LIN {X 0,Y 412.505,Z 413.678,A -85,B 0,C 180,E1 -10494.601,E2 -10494.601} C_VEL
LIN {X 0,Y 412.069,Z 420.208,A -85,B 0,C 180,E1 -10498.081,E2 -10498.081} C_VEL
LIN {X 0,Y 411.614,Z 426.756,A -85,B 0,C 180,E1 -10501.44,E2 -10501.44} C_VEL
LIN {X 0,Y 411.176,Z 433.807,A -85,B 0,C 180,E1 -10504.945,E2 -10504.945} C_VEL
LIN {X 0,Y 410.804,Z 440.902,A -85,B 0,C 180,E1 -10508.419,E2 -10508.419} C_VEL
LIN {X 0,Y 410.512,Z 447.336,A -85,B 0,C 180,E1 -10511.535,E2 -10511.535} C_VEL
LIN {X 0,Y 410.473,Z 449.297,A -85,B 0,C 180,E1 -10512.42,E2 -10512.42} C_VEL
LIN {X 0,Y 412.911,Z 462.619,A -85,B 0,C 180,E1 -10512.936,E2 -10512.936} C_VEL
LIN {X 0,Y 414.711,Z 476.29,A -85,B 0,C 180,E1 -10513.666,E2 -10513.666} C_VEL
LIN {X 0,Y 414.65,Z 482.208,A -85,B 0,C 180,E1 -10514.024,E2 -10514.024} C_VEL
LIN {X 0,Y 413.868,Z 493.865,A -85,B 0,C 180,E1 -10514.865,E2 -10514.865} C_VEL
LIN {X 0,Y 413.021,Z 505.142,A -85,B 0,C 180,E1 -10515.911,E2 -10515.911} C_VEL
LIN {X 0,Y 412.454,Z 514.201,A -85,B 0,C 180,E1 -10516.952,E2 -10516.952} C_VEL
LIN {X 0,Y 411.692,Z 523.047,A -85,B 0,C 180,E1 -10518.179,E2 -10518.179} C_VEL
LIN {X 0,Y 411.033,Z 531.675,A -85,B 0,C 180,E1 -10519.657,E2 -10519.657} C_VEL
LIN {X 0,Y 410.551,Z 538.575,A -85,B 0,C 180,E1 -10521.137,E2 -10521.137} C_VEL
LIN {X 0,Y 410.211,Z 544.105,A -85,B 0,C 180,E1 -10522.617,E2 -10522.617} C_VEL
LIN {X 0,Y 410.036,Z 548.444,A -85,B 0,C 180,E1 -10524.097,E2 -10524.097} C_VEL
LIN {X 0,Y 410.024,Z 550.743,A -85,B 0,C 180,E1 -10525.083,E2 -10525.083} C_VEL
LIN {X 0,Y 409.935,Z 552.604,A -85,B 0,C 180,E1 -10526.068,E2 -10526.068} C_VEL
LIN {X 0,Y 409.967,Z 554.999,A -85,B 0,C 180,E1 -10528.035,E2 -10528.035} C_VEL
LIN {X 0,Y 409.935,Z 555.607,A -85,B 0,C 180,E1 -10529.018,E2 -10529.018} C_VEL
LIN {X 0,Y 409.926,Z 555.822,A -85,B 0,C 180,E1 -10530,E2 -10530} C_VEL
LIN {X 0,Y 409.935,Z 555.605,A -85,B 0,C 180,E1 -10530.982,E2 -10530.982} C_VEL
LIN {X 0,Y 409.967,Z 554.998,A -85,B 0,C 180,E1 -10531.965,E2 -10531.965} C_VEL
LIN {X 0,Y 409.927,Z 553.999,A -85,B 0,C 180,E1 -10532.948,E2 -10532.948} C_VEL
LIN {X 0,Y 409.934,Z 552.601,A -85,B 0,C 180,E1 -10533.932,E2 -10533.932} C_VEL
LIN {X 0,Y 410.025,Z 549.663,A -85,B 0,C 180,E1 -10535.409,E2 -10535.409} C_VEL
LIN {X 0,Y 410.169,Z 545.685,A -85,B 0,C 180,E1 -10536.889,E2 -10536.889} C_VEL
LIN {X 0,Y 410.492,Z 539.57,A -85,B 0,C 180,E1 -10538.616,E2 -10538.616} C_VEL
LIN {X 0,Y 410.934,Z 532.89,A -85,B 0,C 180,E1 -10540.096,E2 -10540.096} C_VEL
LIN {X 0,Y 411.552,Z 524.604,A -85,B 0,C 180,E1 -10541.575,E2 -10541.575} C_VEL
LIN {X 0,Y 412.257,Z 516.113,A -85,B 0,C 180,E1 -10542.804,E2 -10542.804} C_VEL
LIN {X 0,Y 412.969,Z 506.149,A -85,B 0,C 180,E1 -10543.978,E2 -10543.978} C_VEL
LIN {X 0,Y 413.758,Z 495.239,A -85,B 0,C 180,E1 -10545.013,E2 -10545.013} C_VEL
LIN {X 0,Y 414.476,Z 483.946,A -85,B 0,C 180,E1 -10545.862,E2 -10545.862} C_VEL
LIN {X 0,Y 414.712,Z 476.208,A -85,B 0,C 180,E1 -10546.333,E2 -10546.333} C_VEL
LIN {X 0,Y 412.972,Z 463.345,A -85,B 0,C 180,E1 -10547.025,E2 -10547.025} C_VEL
LIN {X 0,Y 410.672,Z 450.687,A -85,B 0,C 180,E1 -10547.534,E2 -10547.534} C_VEL
LIN {X 0,Y 410.438,Z 449.15,A -85,B 0,C 180,E1 -10547.581,E2 -10547.581} C_VEL
LIN {X 0,Y 410.775,Z 441.97,A -85,B 0,C 180,E1 -10551.057,E2 -10551.057} C_VEL
LIN {X 0,Y 411.043,Z 435.469,A -85,B 0,C 180,E1 -10554.227,E2 -10554.227} C_VEL
LIN {X 0,Y 411.426,Z 428.914,A -85,B 0,C 180,E1 -10557.466,E2 -10557.466} C_VEL
LIN {X 0,Y 411.847,Z 423.443,A -85,B 0,C 180,E1 -10560.226,E2 -10560.226} C_VEL
LIN {X 0,Y 412.237,Z 417.454,A -85,B 0,C 180,E1 -10563.345,E2 -10563.345} C_VEL
LIN {X 0,Y 412.438,Z 412.57,A -85,B 0,C 180,E1 -10566.007,E2 -10566.007} C_VEL
LIN {X 0,Y 412.03,Z 408.565,A -85,B 0,C 180,E1 -10568.314,E2 -10568.314} C_VEL
LIN {X 0,Y 411.234,Z 404.262,A -85,B 0,C 180,E1 -10571.068,E2 -10571.068} C_VEL
LIN {X 0,Y 411.181,Z 404.267,A -85,B 0,C 180,E1 -10574.49,E2 -10574.49} C_VEL
LIN {X 0,Y 411.178,Z 404.264,A -85,B 0,C 180,E1 -10578.195,E2 -10578.195} C_VEL
LIN {X 0,Y 411.223,Z 404.263,A -85,B 0,C 180,E1 -10580.776,E2 -10580.776} C_VEL
LIN {X 0,Y 411.201,Z 404.264,A -85,B 0,C 180,E1 -10584.471,E2 -10584.471} C_VEL
LIN {X 0,Y 411.208,Z 404.265,A -85,B 0,C 180,E1 -10586.873,E2 -10586.873} C_VEL
LIN {X 0,Y 411.234,Z 404.261,A -85,B 0,C 180,E1 -10590.644,E2 -10590.644} C_VEL
LIN {X 0,Y 411.238,Z 404.257,A -85,B 0,C 180,E1 -10593.619,E2 -10593.619} C_VEL
LIN {X 0,Y 411.203,Z 404.265,A -85,B 0,C 180,E1 -10596.852,E2 -10596.852} C_VEL
LIN {X 0,Y 411.217,Z 404.262,A -85,B 0,C 180,E1 -10600.05,E2 -10600.05} C_VEL
LIN {X 0,Y 411.264,Z 404.255,A -85,B 0,C 180,E1 -10603.131,E2 -10603.131} C_VEL
LIN {X 0,Y 411.315,Z 404.25,A -85,B 0,C 180,E1 -10606.891,E2 -10606.891} C_VEL
LIN {X 0,Y 411.31,Z 404.253,A -85,B 0,C 180,E1 -10610.162,E2 -10610.162} C_VEL
LIN {X 0,Y 411.462,Z 404.23,A -85,B 0,C 180,E1 -10613.133,E2 -10613.133} C_VEL
LIN {X 0,Y 411.311,Z 404.248,A -85,B 0,C 180,E1 -10615.099,E2 -10615.099} C_VEL
LIN {X 0,Y 411.513,Z 404.226,A -85,B 0,C 180,E1 -10618.043,E2 -10618.043} C_VEL
LIN {X 0,Y 411.644,Z 404.21,A -85,B 0,C 180,E1 -10620,E2 -10620} C_VEL
LIN {X 0,Y 411.459,Z 404.23,A -85,B 0,C 180,E1 -10622.937,E2 -10622.937} C_VEL
LIN {X 0,Y 411.463,Z 404.23,A -85,B 0,C 180,E1 -10626.867,E2 -10626.867} C_VEL
LIN {X 0,Y 411.31,Z 404.251,A -85,B 0,C 180,E1 -10629.838,E2 -10629.838} C_VEL
LIN {X 0,Y 411.315,Z 404.247,A -85,B 0,C 180,E1 -10633.109,E2 -10633.109} C_VEL
LIN {X 0,Y 411.259,Z 404.255,A -85,B 0,C 180,E1 -10636.889,E2 -10636.889} C_VEL
LIN {X 0,Y 411.232,Z 404.262,A -85,B 0,C 180,E1 -10639.987,E2 -10639.987} C_VEL
LIN {X 0,Y 411.204,Z 404.262,A -85,B 0,C 180,E1 -10643.148,E2 -10643.148} C_VEL
LIN {X 0,Y 411.238,Z 404.257,A -85,B 0,C 180,E1 -10646.381,E2 -10646.381} C_VEL
LIN {X 0,Y 411.202,Z 404.266,A -85,B 0,C 180,E1 -10649.713,E2 -10649.713} C_VEL
LIN {X 0,Y 411.208,Z 404.264,A -85,B 0,C 180,E1 -10653.156,E2 -10653.156} C_VEL
LIN {X 0,Y 411.197,Z 404.262,A -85,B 0,C 180,E1 -10656.553,E2 -10656.553} C_VEL
LIN {X 0,Y 411.22,Z 404.262,A -85,B 0,C 180,E1 -10659.729,E2 -10659.729} C_VEL
LIN {X 0,Y 411.175,Z 404.269,A -85,B 0,C 180,E1 -10663.134,E2 -10663.134} C_VEL
LIN {X 0,Y 411.174,Z 404.267,A -85,B 0,C 180,E1 -10665.88,E2 -10665.88} C_VEL
LIN {X 0,Y 411.166,Z 404.268,A -85,B 0,C 180,E1 -10668.772,E2 -10668.772} C_VEL
LIN {X 0,Y 411.203,Z 404.266,A -85,B 0,C 180,E1 -10671.832,E2 -10671.832} C_VEL
LIN {X 0,Y 411.062,Z 404.442,A -85,B 0,C 180,E1 -10674.458,E2 -10674.458} C_VEL
LIN {X 0,Y 411.062,Z 407.378,A -85,B 0,C 180,E1 -10676.905,E2 -10676.905} C_VEL
LIN {X 0,Y 410.847,Z 411.553,A -85,B 0,C 180,E1 -10680.259,E2 -10680.259} C_VEL
LIN {X 0,Y 410.656,Z 415.795,A -85,B 0,C 180,E1 -10683.579,E2 -10683.579} C_VEL
LIN {X 0,Y 410.558,Z 418.639,A -85,B 0,C 180,E1 -10685.743,E2 -10685.743} C_VEL
LIN {X 0,Y 410.376,Z 422.946,A -85,B 0,C 180,E1 -10688.922,E2 -10688.922} C_VEL
LIN {X 0,Y 410.291,Z 427.335,A -85,B 0,C 180,E1 -10692.042,E2 -10692.042} C_VEL
LIN {X 0,Y 410.305,Z 428.198,A -85,B 0,C 180,E1 -10692.495,E2 -10692.495} C_VEL
LIN {X 0,Y 413.403,Z 441.217,A -85,B 0,C 180,E1 -10693.063,E2 -10693.063} C_VEL
LIN {X 0,Y 415.297,Z 451.396,A -85,B 0,C 180,E1 -10693.628,E2 -10693.628} C_VEL
LIN {X 0,Y 414.751,Z 463.825,A -85,B 0,C 180,E1 -10694.395,E2 -10694.395} C_VEL
LIN {X 0,Y 414.051,Z 474.588,A -85,B 0,C 180,E1 -10695.25,E2 -10695.25} C_VEL
LIN {X 0,Y 413.366,Z 485.554,A -85,B 0,C 180,E1 -10696.355,E2 -10696.355} C_VEL
LIN {X 0,Y 412.581,Z 494.46,A -85,B 0,C 180,E1 -10697.456,E2 -10697.456} C_VEL
LIN {X 0,Y 412.005,Z 502.624,A -85,B 0,C 180,E1 -10698.687,E2 -10698.687} C_VEL
LIN {X 0,Y 411.336,Z 510.624,A -85,B 0,C 180,E1 -10700.162,E2 -10700.162} C_VEL
LIN {X 0,Y 410.76,Z 517.048,A -85,B 0,C 180,E1 -10701.638,E2 -10701.638} C_VEL
LIN {X 0,Y 410.435,Z 522.648,A -85,B 0,C 180,E1 -10703.293,E2 -10703.293} C_VEL
LIN {X 0,Y 410.165,Z 527.155,A -85,B 0,C 180,E1 -10705.085,E2 -10705.085} C_VEL
LIN {X 0,Y 410.058,Z 529.016,A -85,B 0,C 180,E1 -10706.069,E2 -10706.069} C_VEL
LIN {X 0,Y 410.06,Z 530.414,A -85,B 0,C 180,E1 -10707.053,E2 -10707.053} C_VEL
LIN {X 0,Y 410.013,Z 531.41,A -85,B 0,C 180,E1 -10708.036,E2 -10708.036} C_VEL
LIN {X 0,Y 409.927,Z 532.258,A -85,B 0,C 180,E1 -10710,E2 -10710} C_VEL
LIN {X 0,Y 409.939,Z 532.07,A -85,B 0,C 180,E1 -10710.982,E2 -10710.982} C_VEL
LIN {X 0,Y 410.013,Z 531.484,A -85,B 0,C 180,E1 -10711.965,E2 -10711.965} C_VEL
LIN {X 0,Y 410.056,Z 530.518,A -85,B 0,C 180,E1 -10712.947,E2 -10712.947} C_VEL
LIN {X 0,Y 410.046,Z 529.165,A -85,B 0,C 180,E1 -10713.931,E2 -10713.931} C_VEL
LIN {X 0,Y 410.272,Z 526.298,A -85,B 0,C 180,E1 -10715.406,E2 -10715.406} C_VEL
LIN {X 0,Y 410.436,Z 522.415,A -85,B 0,C 180,E1 -10716.884,E2 -10716.884} C_VEL
LIN {X 0,Y 410.757,Z 517.403,A -85,B 0,C 180,E1 -10718.363,E2 -10718.363} C_VEL
LIN {X 0,Y 410.982,Z 514.645,A -85,B 0,C 180,E1 -10719.047,E2 -10719.047} C_VEL
LIN {X 0,Y 410.578,Z 511.665,A -85,B 0,C 180,E1 -10719.758,E2 -10719.758} C_VEL
LIN {X 0,Y 408.165,Z 506.457,A -85,B 0,C 180,E1 -10720.893,E2 -10720.893} C_VEL
LIN {X 0,Y 405.817,Z 500.596,A -85,B 0,C 180,E1 -10721.972,E2 -10721.972} C_VEL
LIN {X 0,Y 405.513,Z 496.593,A -85,B 0,C 180,E1 -10722.586,E2 -10722.586} C_VEL
LIN {X 0,Y 406.42,Z 486.565,A -85,B 0,C 180,E1 -10723.883,E2 -10723.883} C_VEL
LIN {X 0,Y 407.086,Z 475.827,A -85,B 0,C 180,E1 -10725.009,E2 -10725.009} C_VEL
LIN {X 0,Y 407.854,Z 465.354,A -85,B 0,C 180,E1 -10725.876,E2 -10725.876} C_VEL
LIN {X 0,Y 408.536,Z 453.254,A -85,B 0,C 180,E1 -10726.654,E2 -10726.654} C_VEL
LIN {X 0,Y 406.632,Z 442.722,A -85,B 0,C 180,E1 -10727.27,E2 -10727.27} C_VEL
LIN {X 0,Y 403.464,Z 429.728,A -85,B 0,C 180,E1 -10727.873,E2 -10727.873} C_VEL
LIN {X 0,Y 403.203,Z 428.147,A -85,B 0,C 180,E1 -10727.947,E2 -10727.947} C_VEL
LIN {X 0,Y 403.303,Z 424.709,A -85,B 0,C 180,E1 -10730.397,E2 -10730.397} C_VEL
LIN {X 0,Y 403.447,Z 420.388,A -85,B 0,C 180,E1 -10733.619,E2 -10733.619} C_VEL
LIN {X 0,Y 403.665,Z 416.097,A -85,B 0,C 180,E1 -10736.915,E2 -10736.915} C_VEL
LIN {X 0,Y 403.841,Z 411.84,A -85,B 0,C 180,E1 -10740.311,E2 -10740.311} C_VEL
LIN {X 0,Y 404.038,Z 407.549,A -85,B 0,C 180,E1 -10743.823,E2 -10743.823} C_VEL
LIN {X 0,Y 404.047,Z 405.966,A -85,B 0,C 180,E1 -10745.162,E2 -10745.162} C_VEL
LIN {X 0,Y 404.083,Z 405.153,A -85,B 0,C 180,E1 -10746.253,E2 -10746.253} C_VEL
LIN {X 0,Y 404.155,Z 405.145,A -85,B 0,C 180,E1 -10748.757,E2 -10748.757} C_VEL
LIN {X 0,Y 404.127,Z 405.143,A -85,B 0,C 180,E1 -10751.6,E2 -10751.6} C_VEL
LIN {X 0,Y 404.151,Z 405.144,A -85,B 0,C 180,E1 -10754.523,E2 -10754.523} C_VEL
LIN {X 0,Y 404.139,Z 405.142,A -85,B 0,C 180,E1 -10757.296,E2 -10757.296} C_VEL
LIN {X 0,Y 404.171,Z 405.137,A -85,B 0,C 180,E1 -10759.955,E2 -10759.955} C_VEL
LIN {X 0,Y 404.142,Z 405.142,A -85,B 0,C 180,E1 -10763.124,E2 -10763.124} C_VEL
LIN {X 0,Y 404.148,Z 405.144,A -85,B 0,C 180,E1 -10766.188,E2 -10766.188} C_VEL
LIN {X 0,Y 404.148,Z 405.141,A -85,B 0,C 180,E1 -10769.715,E2 -10769.715} C_VEL
LIN {X 0,Y 404.198,Z 405.134,A -85,B 0,C 180,E1 -10773.123,E2 -10773.123} C_VEL
LIN {X 0,Y 404.179,Z 405.136,A -85,B 0,C 180,E1 -10775.334,E2 -10775.334} C_VEL
LIN {X 0,Y 404.142,Z 405.144,A -85,B 0,C 180,E1 -10778.581,E2 -10778.581} C_VEL
LIN {X 0,Y 404.212,Z 405.135,A -85,B 0,C 180,E1 -10781.762,E2 -10781.762} C_VEL
LIN {X 0,Y 404.209,Z 405.133,A -85,B 0,C 180,E1 -10784.882,E2 -10784.882} C_VEL
LIN {X 0,Y 404.26,Z 405.131,A -85,B 0,C 180,E1 -10787.959,E2 -10787.959} C_VEL
LIN {X 0,Y 404.436,Z 405.108,A -85,B 0,C 180,E1 -10792.1,E2 -10792.1} C_VEL
LIN {X 0,Y 404.427,Z 405.11,A -85,B 0,C 180,E1 -10794.015,E2 -10794.015} C_VEL
LIN {X 0,Y 404.483,Z 405.104,A -85,B 0,C 180,E1 -10798.008,E2 -10798.008} C_VEL
LIN {X 0,Y 404.613,Z 405.086,A -85,B 0,C 180,E1 -10800,E2 -10800} C_VEL
LIN {X 0,Y 404.419,Z 405.106,A -85,B 0,C 180,E1 -10802.988,E2 -10802.988} C_VEL
LIN {X 0,Y 404.415,Z 405.108,A -85,B 0,C 180,E1 -10806.987,E2 -10806.987} C_VEL
LIN {X 0,Y 404.274,Z 405.127,A -85,B 0,C 180,E1 -10810.011,E2 -10810.011} C_VEL
LIN {X 0,Y 404.269,Z 405.128,A -85,B 0,C 180,E1 -10813.211,E2 -10813.211} C_VEL
LIN {X 0,Y 404.219,Z 405.133,A -85,B 0,C 180,E1 -10817.007,E2 -10817.007} C_VEL
LIN {X 0,Y 404.167,Z 405.138,A -85,B 0,C 180,E1 -10820.351,E2 -10820.351} C_VEL
LIN {X 0,Y 404.171,Z 405.142,A -85,B 0,C 180,E1 -10823.574,E2 -10823.574} C_VEL
LIN {X 0,Y 404.186,Z 405.137,A -85,B 0,C 180,E1 -10825.766,E2 -10825.766} C_VEL
LIN {X 0,Y 404.198,Z 405.133,A -85,B 0,C 180,E1 -10828,E2 -10828} C_VEL
LIN {X 0,Y 404.142,Z 405.144,A -85,B 0,C 180,E1 -10831.558,E2 -10831.558} C_VEL
LIN {X 0,Y 404.188,Z 405.14,A -85,B 0,C 180,E1 -10835.016,E2 -10835.016} C_VEL
LIN {X 0,Y 404.16,Z 405.142,A -85,B 0,C 180,E1 -10838.756,E2 -10838.756} C_VEL
LIN {X 0,Y 404.125,Z 405.143,A -85,B 0,C 180,E1 -10841.6,E2 -10841.6} C_VEL
LIN {X 0,Y 404.149,Z 405.146,A -85,B 0,C 180,E1 -10844.522,E2 -10844.522} C_VEL
LIN {X 0,Y 404.142,Z 405.146,A -85,B 0,C 180,E1 -10847.296,E2 -10847.296} C_VEL
LIN {X 0,Y 404.187,Z 405.177,A -85,B 0,C 180,E1 -10848.806,E2 -10848.806} C_VEL
LIN {X 0,Y 405.069,Z 410.343,A -85,B 0,C 180,E1 -10851.996,E2 -10851.996} C_VEL
LIN {X 0,Y 405.49,Z 414.727,A -85,B 0,C 180,E1 -10854.549,E2 -10854.549} C_VEL
LIN {X 0,Y 405.09,Z 420.075,A -85,B 0,C 180,E1 -10857.464,E2 -10857.464} C_VEL
LIN {X 0,Y 404.623,Z 426.609,A -85,B 0,C 180,E1 -10860.9,E2 -10860.9} C_VEL
LIN {X 0,Y 404.131,Z 434.138,A -85,B 0,C 180,E1 -10864.73,E2 -10864.73} C_VEL
LIN {X 0,Y 403.798,Z 440.721,A -85,B 0,C 180,E1 -10868.025,E2 -10868.025} C_VEL
LIN {X 0,Y 403.465,Z 447.137,A -85,B 0,C 180,E1 -10871.201,E2 -10871.201} C_VEL
LIN {X 0,Y 403.385,Z 449.094,A -85,B 0,C 180,E1 -10872.101,E2 -10872.101} C_VEL
LIN {X 0,Y 405.927,Z 462.554,A -85,B 0,C 180,E1 -10872.639,E2 -10872.639} C_VEL
LIN {X 0,Y 407.681,Z 475.737,A -85,B 0,C 180,E1 -10873.356,E2 -10873.356} C_VEL
LIN {X 0,Y 407.877,Z 480.462,A -85,B 0,C 180,E1 -10873.652,E2 -10873.652} C_VEL
LIN {X 0,Y 407.117,Z 492.128,A -85,B 0,C 180,E1 -10874.48,E2 -10874.48} C_VEL
LIN {X 0,Y 406.319,Z 502.235,A -85,B 0,C 180,E1 -10875.385,E2 -10875.385} C_VEL
LIN {X 0,Y 405.565,Z 512.037,A -85,B 0,C 180,E1 -10876.471,E2 -10876.471} C_VEL
LIN {X 0,Y 404.869,Z 521.211,A -85,B 0,C 180,E1 -10877.723,E2 -10877.723} C_VEL
LIN {X 0,Y 404.05,Z 530.148,A -85,B 0,C 180,E1 -10879.223,E2 -10879.223} C_VEL
LIN {X 0,Y 403.562,Z 537.345,A -85,B 0,C 180,E1 -10880.73,E2 -10880.73} C_VEL
LIN {X 0,Y 403.288,Z 542.205,A -85,B 0,C 180,E1 -10881.986,E2 -10881.986} C_VEL
LIN {X 0,Y 402.958,Z 547.747,A -85,B 0,C 180,E1 -10883.795,E2 -10883.795} C_VEL
LIN {X 0,Y 402.936,Z 550.539,A -85,B 0,C 180,E1 -10884.997,E2 -10884.997} C_VEL
LIN {X 0,Y 402.855,Z 552.401,A -85,B 0,C 180,E1 -10885.998,E2 -10885.998} C_VEL
LIN {X 0,Y 402.865,Z 554.795,A -85,B 0,C 180,E1 -10888,E2 -10888} C_VEL
LIN {X 0,Y 402.862,Z 555.403,A -85,B 0,C 180,E1 -10889,E2 -10889} C_VEL
LIN {X 0,Y 402.851,Z 555.619,A -85,B 0,C 180,E1 -10890,E2 -10890} C_VEL
LIN {X 0,Y 402.862,Z 555.402,A -85,B 0,C 180,E1 -10890.999,E2 -10890.999} C_VEL
LIN {X 0,Y 402.865,Z 554.793,A -85,B 0,C 180,E1 -10891.999,E2 -10891.999} C_VEL
LIN {X 0,Y 402.855,Z 552.397,A -85,B 0,C 180,E1 -10894.001,E2 -10894.001} C_VEL
LIN {X 0,Y 402.926,Z 549.457,A -85,B 0,C 180,E1 -10895.505,E2 -10895.505} C_VEL
LIN {X 0,Y 403.082,Z 545.479,A -85,B 0,C 180,E1 -10897.01,E2 -10897.01} C_VEL
LIN {X 0,Y 403.43,Z 539.364,A -85,B 0,C 180,E1 -10898.768,E2 -10898.768} C_VEL
LIN {X 0,Y 403.926,Z 532.684,A -85,B 0,C 180,E1 -10900.273,E2 -10900.273} C_VEL
LIN {X 0,Y 404.582,Z 524.397,A -85,B 0,C 180,E1 -10901.777,E2 -10901.777} C_VEL
LIN {X 0,Y 405.298,Z 515.905,A -85,B 0,C 180,E1 -10903.028,E2 -10903.028} C_VEL
LIN {X 0,Y 406.068,Z 505.648,A -85,B 0,C 180,E1 -10904.252,E2 -10904.252} C_VEL
LIN {X 0,Y 406.886,Z 495.031,A -85,B 0,C 180,E1 -10905.272,E2 -10905.272} C_VEL
LIN {X 0,Y 407.627,Z 483.843,A -85,B 0,C 180,E1 -10906.128,E2 -10906.128} C_VEL
LIN {X 0,Y 407.959,Z 478.604,A -85,B 0,C 180,E1 -10906.458,E2 -10906.458} C_VEL
LIN {X 0,Y 406.445,Z 465.955,A -85,B 0,C 180,E1 -10907.187,E2 -10907.187} C_VEL
LIN {X 0,Y 404.155,Z 452.998,A -85,B 0,C 180,E1 -10907.755,E2 -10907.755} C_VEL
LIN {X 0,Y 403.394,Z 448.919,A -85,B 0,C 180,E1 -10907.915,E2 -10907.915} C_VEL
LIN {X 0,Y 403.717,Z 441.782,A -85,B 0,C 180,E1 -10911.443,E2 -10911.443} C_VEL
LIN {X 0,Y 404.034,Z 435.299,A -85,B 0,C 180,E1 -10914.675,E2 -10914.675} C_VEL
LIN {X 0,Y 404.449,Z 428.754,A -85,B 0,C 180,E1 -10917.981,E2 -10917.981} C_VEL
LIN {X 0,Y 404.86,Z 423.297,A -85,B 0,C 180,E1 -10920.803,E2 -10920.803} C_VEL
LIN {X 0,Y 405.331,Z 416.772,A -85,B 0,C 180,E1 -10924.299,E2 -10924.299} C_VEL
LIN {X 0,Y 405.424,Z 413.536,A -85,B 0,C 180,E1 -10926.114,E2 -10926.114} C_VEL
LIN {X 0,Y 404.922,Z 409.208,A -85,B 0,C 180,E1 -10928.67,E2 -10928.67} C_VEL
LIN {X 0,Y 404.171,Z 405.142,A -85,B 0,C 180,E1 -10931.278,E2 -10931.278} C_VEL
LIN {X 0,Y 404.15,Z 405.142,A -85,B 0,C 180,E1 -10934.523,E2 -10934.523} C_VEL
LIN {X 0,Y 404.138,Z 405.145,A -85,B 0,C 180,E1 -10937.296,E2 -10937.296} C_VEL
LIN {X 0,Y 404.17,Z 405.137,A -85,B 0,C 180,E1 -10939.955,E2 -10939.955} C_VEL
LIN {X 0,Y 404.141,Z 405.145,A -85,B 0,C 180,E1 -10943.124,E2 -10943.124} C_VEL
LIN {X 0,Y 404.146,Z 405.141,A -85,B 0,C 180,E1 -10946.188,E2 -10946.188} C_VEL
LIN {X 0,Y 404.147,Z 405.14,A -85,B 0,C 180,E1 -10949.715,E2 -10949.715} C_VEL
LIN {X 0,Y 404.196,Z 405.137,A -85,B 0,C 180,E1 -10953.123,E2 -10953.123} C_VEL
LIN {X 0,Y 404.178,Z 405.138,A -85,B 0,C 180,E1 -10955.334,E2 -10955.334} C_VEL
LIN {X 0,Y 404.14,Z 405.145,A -85,B 0,C 180,E1 -10958.581,E2 -10958.581} C_VEL
LIN {X 0,Y 404.212,Z 405.132,A -85,B 0,C 180,E1 -10961.762,E2 -10961.762} C_VEL
LIN {X 0,Y 404.21,Z 405.134,A -85,B 0,C 180,E1 -10964.882,E2 -10964.882} C_VEL
LIN {X 0,Y 404.272,Z 405.126,A -85,B 0,C 180,E1 -10967.959,E2 -10967.959} C_VEL
LIN {X 0,Y 404.435,Z 405.109,A -85,B 0,C 180,E1 -10972.1,E2 -10972.1} C_VEL
LIN {X 0,Y 404.426,Z 405.109,A -85,B 0,C 180,E1 -10974.015,E2 -10974.015} C_VEL
LIN {X 0,Y 404.482,Z 405.102,A -85,B 0,C 180,E1 -10978.009,E2 -10978.009} C_VEL
LIN {X 0,Y 404.614,Z 405.086,A -85,B 0,C 180,E1 -10980,E2 -10980} C_VEL
LIN {X 0,Y 404.417,Z 405.107,A -85,B 0,C 180,E1 -10982.988,E2 -10982.988} C_VEL
LIN {X 0,Y 404.414,Z 405.107,A -85,B 0,C 180,E1 -10986.987,E2 -10986.987} C_VEL
LIN {X 0,Y 404.273,Z 405.129,A -85,B 0,C 180,E1 -10990.011,E2 -10990.011} C_VEL
LIN {X 0,Y 404.268,Z 405.125,A -85,B 0,C 180,E1 -10993.211,E2 -10993.211} C_VEL
LIN {X 0,Y 404.217,Z 405.132,A -85,B 0,C 180,E1 -10997.007,E2 -10997.007} C_VEL
LIN {X 0,Y 404.165,Z 405.14,A -85,B 0,C 180,E1 -11000.352,E2 -11000.352} C_VEL
LIN {X 0,Y 404.17,Z 405.141,A -85,B 0,C 180,E1 -11003.575,E2 -11003.575} C_VEL
LIN {X 0,Y 404.185,Z 405.141,A -85,B 0,C 180,E1 -11005.767,E2 -11005.767} C_VEL
LIN {X 0,Y 404.197,Z 405.137,A -85,B 0,C 180,E1 -11008,E2 -11008} C_VEL
LIN {X 0,Y 404.141,Z 405.145,A -85,B 0,C 180,E1 -11011.558,E2 -11011.558} C_VEL
LIN {X 0,Y 404.187,Z 405.137,A -85,B 0,C 180,E1 -11015.016,E2 -11015.016} C_VEL
LIN {X 0,Y 404.161,Z 405.138,A -85,B 0,C 180,E1 -11018.756,E2 -11018.756} C_VEL
LIN {X 0,Y 404.125,Z 405.147,A -85,B 0,C 180,E1 -11021.6,E2 -11021.6} C_VEL
LIN {X 0,Y 404.148,Z 405.141,A -85,B 0,C 180,E1 -11024.522,E2 -11024.522} C_VEL
LIN {X 0,Y 404.141,Z 405.145,A -85,B 0,C 180,E1 -11027.296,E2 -11027.296} C_VEL
LIN {X 0,Y 404.171,Z 405.138,A -85,B 0,C 180,E1 -11029.956,E2 -11029.956} C_VEL
LIN {X 0,Y 404.114,Z 405.15,A -85,B 0,C 180,E1 -11033.13,E2 -11033.13} C_VEL
LIN {X 0,Y 404.084,Z 405.153,A -85,B 0,C 180,E1 -11033.748,E2 -11033.748} C_VEL
LIN {X 0,Y 404.053,Z 406,A -85,B 0,C 180,E1 -11034.971,E2 -11034.971} C_VEL
LIN {X 0,Y 403.979,Z 408.859,A -85,B 0,C 180,E1 -11037.364,E2 -11037.364} C_VEL
LIN {X 0,Y 403.781,Z 413.122,A -85,B 0,C 180,E1 -11040.833,E2 -11040.833} C_VEL
LIN {X 0,Y 403.56,Z 417.373,A -85,B 0,C 180,E1 -11044.191,E2 -11044.191} C_VEL
LIN {X 0,Y 403.383,Z 421.689,A -85,B 0,C 180,E1 -11047.462,E2 -11047.462} C_VEL
LIN {X 0,Y 403.293,Z 426.05,A -85,B 0,C 180,E1 -11050.664,E2 -11050.664} C_VEL
LIN {X 0,Y 403.24,Z 428.168,A -85,B 0,C 180,E1 -11052.168,E2 -11052.168} C_VEL
LIN {X 0,Y 406.5,Z 441.982,A -85,B 0,C 180,E1 -11052.79,E2 -11052.79} C_VEL
LIN {X 0,Y 408.45,Z 452.367,A -85,B 0,C 180,E1 -11053.389,E2 -11053.389} C_VEL
LIN {X 0,Y 407.908,Z 464.036,A -85,B 0,C 180,E1 -11054.126,E2 -11054.126} C_VEL
LIN {X 0,Y 407.194,Z 474.798,A -85,B 0,C 180,E1 -11054.996,E2 -11054.996} C_VEL
LIN {X 0,Y 406.483,Z 485.762,A -85,B 0,C 180,E1 -11056.12,E2 -11056.12} C_VEL
LIN {X 0,Y 405.661,Z 494.667,A -85,B 0,C 180,E1 -11057.239,E2 -11057.239} C_VEL
LIN {X 0,Y 405.018,Z 502.832,A -85,B 0,C 180,E1 -11058.489,E2 -11058.489} C_VEL
LIN {X 0,Y 404.334,Z 510.831,A -85,B 0,C 180,E1 -11059.99,E2 -11059.99} C_VEL
LIN {X 0,Y 403.72,Z 517.254,A -85,B 0,C 180,E1 -11061.491,E2 -11061.491} C_VEL
LIN {X 0,Y 403.347,Z 523.226,A -85,B 0,C 180,E1 -11063.307,E2 -11063.307} C_VEL
LIN {X 0,Y 403.11,Z 527.36,A -85,B 0,C 180,E1 -11064.999,E2 -11064.999} C_VEL
LIN {X 0,Y 402.974,Z 529.22,A -85,B 0,C 180,E1 -11066,E2 -11066} C_VEL
LIN {X 0,Y 402.964,Z 530.619,A -85,B 0,C 180,E1 -11067.001,E2 -11067.001} C_VEL
LIN {X 0,Y 402.945,Z 531.613,A -85,B 0,C 180,E1 -11068.001,E2 -11068.001} C_VEL
LIN {X 0,Y 402.851,Z 532.462,A -85,B 0,C 180,E1 -11070,E2 -11070} C_VEL
LIN {X 0,Y 402.867,Z 532.273,A -85,B 0,C 180,E1 -11071,E2 -11071} C_VEL
LIN {X 0,Y 402.945,Z 531.687,A -85,B 0,C 180,E1 -11071.999,E2 -11071.999} C_VEL
LIN {X 0,Y 402.959,Z 530.722,A -85,B 0,C 180,E1 -11072.999,E2 -11072.999} C_VEL
LIN {X 0,Y 402.964,Z 529.368,A -85,B 0,C 180,E1 -11074,E2 -11074} C_VEL
LIN {X 0,Y 403.22,Z 526.501,A -85,B 0,C 180,E1 -11075.501,E2 -11075.501} C_VEL
LIN {X 0,Y 403.395,Z 522.618,A -85,B 0,C 180,E1 -11077.005,E2 -11077.005} C_VEL
LIN {X 0,Y 403.716,Z 517.606,A -85,B 0,C 180,E1 -11078.509,E2 -11078.509} C_VEL
LIN {X 0,Y 404.273,Z 511.293,A -85,B 0,C 180,E1 -11080.011,E2 -11080.011} C_VEL
LIN {X 0,Y 404.926,Z 503.392,A -85,B 0,C 180,E1 -11081.514,E2 -11081.514} C_VEL
LIN {X 0,Y 405.513,Z 496.593,A -85,B 0,C 180,E1 -11082.586,E2 -11082.586} C_VEL
LIN {X 0,Y 405.236,Z 492.479,A -85,B 0,C 180,E1 -11083.178,E2 -11083.178} C_VEL
LIN {X 0,Y 401.987,Z 482.703,A -85,B 0,C 180,E1 -11084.505,E2 -11084.505} C_VEL
LIN {X 0,Y 400.532,Z 476.618,A -85,B 0,C 180,E1 -11085.199,E2 -11085.199} C_VEL
LIN {X 0,Y 400.436,Z 473.331,A -85,B 0,C 180,E1 -11085.514,E2 -11085.514} C_VEL
LIN {X 0,Y 401.37,Z 460.844,A -85,B 0,C 180,E1 -11086.488,E2 -11086.488} C_VEL
LIN {X 0,Y 401.68,Z 454.069,A -85,B 0,C 180,E1 -11086.91,E2 -11086.91} C_VEL
LIN {X 0,Y 399.837,Z 443.933,A -85,B 0,C 180,E1 -11087.529,E2 -11087.529} C_VEL
LIN {X 0,Y 396.657,Z 430.628,A -85,B 0,C 180,E1 -11088.169,E2 -11088.169} C_VEL
LIN {X 0,Y 396.147,Z 428.332,A -85,B 0,C 180,E1 -11088.288,E2 -11088.288} C_VEL
LIN {X 0,Y 396.236,Z 424.898,A -85,B 0,C 180,E1 -11090.778,E2 -11090.778} C_VEL
LIN {X 0,Y 396.429,Z 420.565,A -85,B 0,C 180,E1 -11094.064,E2 -11094.064} C_VEL
LIN {X 0,Y 396.633,Z 416.015,A -85,B 0,C 180,E1 -11097.63,E2 -11097.63} C_VEL
LIN {X 0,Y 396.834,Z 411.989,A -85,B 0,C 180,E1 -11100.904,E2 -11100.904} C_VEL
LIN {X 0,Y 397.009,Z 407.685,A -85,B 0,C 180,E1 -11104.505,E2 -11104.505} C_VEL
LIN {X 0,Y 397.011,Z 406.243,A -85,B 0,C 180,E1 -11105.745,E2 -11105.745} C_VEL
LIN {X 0,Y 397.101,Z 406.022,A -85,B 0,C 180,E1 -11108.275,E2 -11108.275} C_VEL
LIN {X 0,Y 397.092,Z 406.023,A -85,B 0,C 180,E1 -11110.909,E2 -11110.909} C_VEL
LIN {X 0,Y 397.106,Z 406.018,A -85,B 0,C 180,E1 -11113.648,E2 -11113.648} C_VEL
LIN {X 0,Y 397.105,Z 406.022,A -85,B 0,C 180,E1 -11116.521,E2 -11116.521} C_VEL
LIN {X 0,Y 397.117,Z 406.019,A -85,B 0,C 180,E1 -11120.423,E2 -11120.423} C_VEL
LIN {X 0,Y 397.112,Z 406.02,A -85,B 0,C 180,E1 -11124.265,E2 -11124.265} C_VEL
LIN {X 0,Y 397.117,Z 406.02,A -85,B 0,C 180,E1 -11126.727,E2 -11126.727} C_VEL
LIN {X 0,Y 397.127,Z 406.019,A -85,B 0,C 180,E1 -11130.296,E2 -11130.296} C_VEL
LIN {X 0,Y 397.197,Z 406.009,A -85,B 0,C 180,E1 -11132.61,E2 -11132.61} C_VEL
LIN {X 0,Y 397.135,Z 406.016,A -85,B 0,C 180,E1 -11135.982,E2 -11135.982} C_VEL
LIN {X 0,Y 397.142,Z 406.014,A -85,B 0,C 180,E1 -11139.705,E2 -11139.705} C_VEL
LIN {X 0,Y 397.185,Z 406.008,A -85,B 0,C 180,E1 -11142.845,E2 -11142.845} C_VEL
LIN {X 0,Y 397.231,Z 406.002,A -85,B 0,C 180,E1 -11146.703,E2 -11146.703} C_VEL
LIN {X 0,Y 397.221,Z 406.007,A -85,B 0,C 180,E1 -11149.809,E2 -11149.809} C_VEL
LIN {X 0,Y 397.367,Z 405.985,A -85,B 0,C 180,E1 -11152.888,E2 -11152.888} C_VEL
LIN {X 0,Y 397.257,Z 405.999,A -85,B 0,C 180,E1 -11154.925,E2 -11154.925} C_VEL
LIN {X 0,Y 397.452,Z 405.98,A -85,B 0,C 180,E1 -11157.973,E2 -11157.973} C_VEL
LIN {X 0,Y 397.582,Z 405.962,A -85,B 0,C 180,E1 -11160,E2 -11160} C_VEL
LIN {X 0,Y 397.378,Z 405.983,A -85,B 0,C 180,E1 -11163.041,E2 -11163.041} C_VEL
LIN {X 0,Y 397.367,Z 405.986,A -85,B 0,C 180,E1 -11167.112,E2 -11167.112} C_VEL
LIN {X 0,Y 397.232,Z 406.003,A -85,B 0,C 180,E1 -11170.191,E2 -11170.191} C_VEL
LIN {X 0,Y 397.229,Z 406.005,A -85,B 0,C 180,E1 -11173.321,E2 -11173.321} C_VEL
LIN {X 0,Y 397.185,Z 406.01,A -85,B 0,C 180,E1 -11177.155,E2 -11177.155} C_VEL
LIN {X 0,Y 397.105,Z 406.018,A -85,B 0,C 180,E1 -11180.73,E2 -11180.73} C_VEL
LIN {X 0,Y 397.135,Z 406.014,A -85,B 0,C 180,E1 -11184.018,E2 -11184.018} C_VEL
LIN {X 0,Y 397.197,Z 406.011,A -85,B 0,C 180,E1 -11187.39,E2 -11187.39} C_VEL
LIN {X 0,Y 397.081,Z 406.023,A -85,B 0,C 180,E1 -11190.882,E2 -11190.882} C_VEL
LIN {X 0,Y 397.128,Z 406.016,A -85,B 0,C 180,E1 -11194.493,E2 -11194.493} C_VEL
LIN {X 0,Y 397.108,Z 406.017,A -85,B 0,C 180,E1 -11198.274,E2 -11198.274} C_VEL
LIN {X 0,Y 397.091,Z 406.024,A -85,B 0,C 180,E1 -11200.909,E2 -11200.909} C_VEL
LIN {X 0,Y 397.103,Z 406.02,A -85,B 0,C 180,E1 -11203.648,E2 -11203.648} C_VEL
LIN {X 0,Y 397.107,Z 406.024,A -85,B 0,C 180,E1 -11206.52,E2 -11206.52} C_VEL
LIN {X 0,Y 397.143,Z 406.159,A -85,B 0,C 180,E1 -11208.593,E2 -11208.593} C_VEL
LIN {X 0,Y 398.048,Z 411.281,A -85,B 0,C 180,E1 -11211.832,E2 -11211.832} C_VEL
LIN {X 0,Y 398.466,Z 415.607,A -85,B 0,C 180,E1 -11214.405,E2 -11214.405} C_VEL
LIN {X 0,Y 398.065,Z 421.018,A -85,B 0,C 180,E1 -11217.419,E2 -11217.419} C_VEL
LIN {X 0,Y 397.583,Z 427.538,A -85,B 0,C 180,E1 -11220.914,E2 -11220.914} C_VEL
LIN {X 0,Y 397.07,Z 435.155,A -85,B 0,C 180,E1 -11224.862,E2 -11224.862} C_VEL
LIN {X 0,Y 396.695,Z 441.62,A -85,B 0,C 180,E1 -11228.158,E2 -11228.158} C_VEL
LIN {X 0,Y 396.324,Z 448.735,A -85,B 0,C 180,E1 -11231.754,E2 -11231.754} C_VEL
LIN {X 0,Y 399.047,Z 463.119,A -85,B 0,C 180,E1 -11232.363,E2 -11232.363} C_VEL
LIN {X 0,Y 400.664,Z 475.154,A -85,B 0,C 180,E1 -11233.034,E2 -11233.034} C_VEL
LIN {X 0,Y 401.032,Z 480.541,A -85,B 0,C 180,E1 -11233.383,E2 -11233.383} C_VEL
LIN {X 0,Y 400.252,Z 491.928,A -85,B 0,C 180,E1 -11234.207,E2 -11234.207} C_VEL
LIN {X 0,Y 399.356,Z 502.911,A -85,B 0,C 180,E1 -11235.216,E2 -11235.216} C_VEL
LIN {X 0,Y 398.529,Z 513.833,A -85,B 0,C 180,E1 -11236.492,E2 -11236.492} C_VEL
LIN {X 0,Y 397.748,Z 522.641,A -85,B 0,C 180,E1 -11237.758,E2 -11237.758} C_VEL
LIN {X 0,Y 396.962,Z 531.267,A -85,B 0,C 180,E1 -11239.286,E2 -11239.286} C_VEL
LIN {X 0,Y 396.451,Z 538.167,A -85,B 0,C 180,E1 -11240.819,E2 -11240.819} C_VEL
LIN {X 0,Y 396.09,Z 543.697,A -85,B 0,C 180,E1 -11242.353,E2 -11242.353} C_VEL
LIN {X 0,Y 395.831,Z 548.779,A -85,B 0,C 180,E1 -11244.189,E2 -11244.189} C_VEL
LIN {X 0,Y 395.778,Z 552.197,A -85,B 0,C 180,E1 -11245.927,E2 -11245.927} C_VEL
LIN {X 0,Y 395.763,Z 554.591,A -85,B 0,C 180,E1 -11247.965,E2 -11247.965} C_VEL
LIN {X 0,Y 395.791,Z 555.2,A -85,B 0,C 180,E1 -11248.982,E2 -11248.982} C_VEL
LIN {X 0,Y 395.778,Z 555.416,A -85,B 0,C 180,E1 -11250,E2 -11250} C_VEL
LIN {X 0,Y 395.791,Z 555.198,A -85,B 0,C 180,E1 -11251.017,E2 -11251.017} C_VEL
LIN {X 0,Y 395.763,Z 554.589,A -85,B 0,C 180,E1 -11252.035,E2 -11252.035} C_VEL
LIN {X 0,Y 395.778,Z 552.192,A -85,B 0,C 180,E1 -11254.073,E2 -11254.073} C_VEL
LIN {X 0,Y 395.831,Z 548.765,A -85,B 0,C 180,E1 -11255.811,E2 -11255.811} C_VEL
LIN {X 0,Y 396.09,Z 543.678,A -85,B 0,C 180,E1 -11257.647,E2 -11257.647} C_VEL
LIN {X 0,Y 396.45,Z 538.144,A -85,B 0,C 180,E1 -11259.18,E2 -11259.18} C_VEL
LIN {X 0,Y 396.961,Z 531.238,A -85,B 0,C 180,E1 -11260.713,E2 -11260.713} C_VEL
LIN {X 0,Y 397.768,Z 522.603,A -85,B 0,C 180,E1 -11262.241,E2 -11262.241} C_VEL
LIN {X 0,Y 398.516,Z 513.783,A -85,B 0,C 180,E1 -11263.508,E2 -11263.508} C_VEL
LIN {X 0,Y 399.328,Z 503.319,A -85,B 0,C 180,E1 -11264.733,E2 -11264.733} C_VEL
LIN {X 0,Y 400.136,Z 493.393,A -85,B 0,C 180,E1 -11265.667,E2 -11265.667} C_VEL
LIN {X 0,Y 400.921,Z 482.137,A -85,B 0,C 180,E1 -11266.509,E2 -11266.509} C_VEL
LIN {X 0,Y 400.858,Z 476.998,A -85,B 0,C 180,E1 -11266.844,E2 -11266.844} C_VEL
LIN {X 0,Y 399.177,Z 464.033,A -85,B 0,C 180,E1 -11267.584,E2 -11267.584} C_VEL
LIN {X 0,Y 396.667,Z 450.681,A -85,B 0,C 180,E1 -11268.163,E2 -11268.163} C_VEL
LIN {X 0,Y 396.323,Z 448.72,A -85,B 0,C 180,E1 -11268.246,E2 -11268.246} C_VEL
LIN {X 0,Y 396.694,Z 441.599,A -85,B 0,C 180,E1 -11271.842,E2 -11271.842} C_VEL
LIN {X 0,Y 397.081,Z 434.451,A -85,B 0,C 180,E1 -11275.49,E2 -11275.49} C_VEL
LIN {X 0,Y 397.711,Z 426.426,A -85,B 0,C 180,E1 -11279.656,E2 -11279.656} C_VEL
LIN {X 0,Y 398.157,Z 419.888,A -85,B 0,C 180,E1 -11283.174,E2 -11283.174} C_VEL
LIN {X 0,Y 398.425,Z 415.279,A -85,B 0,C 180,E1 -11285.765,E2 -11285.765} C_VEL
LIN {X 0,Y 398.069,Z 411.261,A -85,B 0,C 180,E1 -11288.165,E2 -11288.165} C_VEL
LIN {X 0,Y 397.113,Z 406.022,A -85,B 0,C 180,E1 -11291.495,E2 -11291.495} C_VEL
LIN {X 0,Y 397.091,Z 406.024,A -85,B 0,C 180,E1 -11295.068,E2 -11295.068} C_VEL
LIN {X 0,Y 397.067,Z 406.021,A -85,B 0,C 180,E1 -11298.021,E2 -11298.021} C_VEL
LIN {X 0,Y 397.134,Z 406.018,A -85,B 0,C 180,E1 -11301.138,E2 -11301.138} C_VEL
LIN {X 0,Y 397.121,Z 406.018,A -85,B 0,C 180,E1 -11304.496,E2 -11304.496} C_VEL
LIN {X 0,Y 397.079,Z 406.021,A -85,B 0,C 180,E1 -11307.928,E2 -11307.928} C_VEL
LIN {X 0,Y 397.123,Z 406.015,A -85,B 0,C 180,E1 -11311.456,E2 -11311.456} C_VEL
LIN {X 0,Y 397.154,Z 406.015,A -85,B 0,C 180,E1 -11314.488,E2 -11314.488} C_VEL
LIN {X 0,Y 397.11,Z 406.019,A -85,B 0,C 180,E1 -11317.086,E2 -11317.086} C_VEL
LIN {X 0,Y 397.15,Z 406.016,A -85,B 0,C 180,E1 -11320.353,E2 -11320.353} C_VEL
LIN {X 0,Y 397.168,Z 406.009,A -85,B 0,C 180,E1 -11323.553,E2 -11323.553} C_VEL
LIN {X 0,Y 397.23,Z 406.005,A -85,B 0,C 180,E1 -11326.703,E2 -11326.703} C_VEL
LIN {X 0,Y 397.23,Z 406.003,A -85,B 0,C 180,E1 -11329.809,E2 -11329.809} C_VEL
LIN {X 0,Y 397.366,Z 405.987,A -85,B 0,C 180,E1 -11332.888,E2 -11332.888} C_VEL
LIN {X 0,Y 397.256,Z 406,A -85,B 0,C 180,E1 -11334.925,E2 -11334.925} C_VEL
LIN {X 0,Y 397.451,Z 405.977,A -85,B 0,C 180,E1 -11337.973,E2 -11337.973} C_VEL
LIN {X 0,Y 397.583,Z 405.961,A -85,B 0,C 180,E1 -11340,E2 -11340} C_VEL
LIN {X 0,Y 397.377,Z 405.984,A -85,B 0,C 180,E1 -11343.041,E2 -11343.041} C_VEL
LIN {X 0,Y 397.366,Z 405.985,A -85,B 0,C 180,E1 -11347.112,E2 -11347.112} C_VEL
LIN {X 0,Y 397.231,Z 406.006,A -85,B 0,C 180,E1 -11350.191,E2 -11350.191} C_VEL
LIN {X 0,Y 397.228,Z 406.002,A -85,B 0,C 180,E1 -11353.321,E2 -11353.321} C_VEL
LIN {X 0,Y 397.183,Z 406.008,A -85,B 0,C 180,E1 -11357.155,E2 -11357.155} C_VEL
LIN {X 0,Y 397.104,Z 406.018,A -85,B 0,C 180,E1 -11360.73,E2 -11360.73} C_VEL
LIN {X 0,Y 397.134,Z 406.017,A -85,B 0,C 180,E1 -11364.018,E2 -11364.018} C_VEL
LIN {X 0,Y 397.196,Z 406.009,A -85,B 0,C 180,E1 -11367.39,E2 -11367.39} C_VEL
LIN {X 0,Y 397.08,Z 406.021,A -85,B 0,C 180,E1 -11370.883,E2 -11370.883} C_VEL
LIN {X 0,Y 397.128,Z 406.015,A -85,B 0,C 180,E1 -11374.493,E2 -11374.493} C_VEL
LIN {X 0,Y 397.109,Z 406.016,A -85,B 0,C 180,E1 -11378.275,E2 -11378.275} C_VEL
LIN {X 0,Y 397.091,Z 406.02,A -85,B 0,C 180,E1 -11380.909,E2 -11380.909} C_VEL
LIN {X 0,Y 397.103,Z 406.022,A -85,B 0,C 180,E1 -11383.649,E2 -11383.649} C_VEL
LIN {X 0,Y 397.106,Z 406.018,A -85,B 0,C 180,E1 -11386.521,E2 -11386.521} C_VEL
LIN {X 0,Y 397.115,Z 406.016,A -85,B 0,C 180,E1 -11390.423,E2 -11390.423} C_VEL
LIN {X 0,Y 397.081,Z 406.024,A -85,B 0,C 180,E1 -11393.003,E2 -11393.003} C_VEL
LIN {X 0,Y 396.97,Z 406.117,A -85,B 0,C 180,E1 -11394.251,E2 -11394.251} C_VEL
LIN {X 0,Y 396.961,Z 409.006,A -85,B 0,C 180,E1 -11396.713,E2 -11396.713} C_VEL
LIN {X 0,Y 396.824,Z 411.856,A -85,B 0,C 180,E1 -11399.096,E2 -11399.096} C_VEL
LIN {X 0,Y 396.632,Z 416.121,A -85,B 0,C 180,E1 -11402.568,E2 -11402.568} C_VEL
LIN {X 0,Y 396.428,Z 420.423,A -85,B 0,C 180,E1 -11405.936,E2 -11405.936} C_VEL
LIN {X 0,Y 396.236,Z 424.763,A -85,B 0,C 180,E1 -11409.223,E2 -11409.223} C_VEL
LIN {X 0,Y 396.173,Z 428.368,A -85,B 0,C 180,E1 -11411.839,E2 -11411.839} C_VEL
LIN {X 0,Y 399.387,Z 441.794,A -85,B 0,C 180,E1 -11412.455,E2 -11412.455} C_VEL
LIN {X 0,Y 401.576,Z 453.261,A -85,B 0,C 180,E1 -11413.136,E2 -11413.136} C_VEL
LIN {X 0,Y 401.101,Z 464.246,A -85,B 0,C 180,E1 -11413.85,E2 -11413.85} C_VEL
LIN {X 0,Y 400.34,Z 475.007,A -85,B 0,C 180,E1 -11414.733,E2 -11414.733} C_VEL
LIN {X 0,Y 399.599,Z 485.97,A -85,B 0,C 180,E1 -11415.876,E2 -11415.876} C_VEL
LIN {X 0,Y 398.744,Z 494.874,A -85,B 0,C 180,E1 -11417.013,E2 -11417.013} C_VEL
LIN {X 0,Y 398.034,Z 503.039,A -85,B 0,C 180,E1 -11418.285,E2 -11418.285} C_VEL
LIN {X 0,Y 397.309,Z 511.038,A -85,B 0,C 180,E1 -11419.811,E2 -11419.811} C_VEL
LIN {X 0,Y 396.696,Z 517.46,A -85,B 0,C 180,E1 -11421.339,E2 -11421.339} C_VEL
LIN {X 0,Y 396.362,Z 522.55,A -85,B 0,C 180,E1 -11422.87,E2 -11422.87} C_VEL
LIN {X 0,Y 396.152,Z 526.502,A -85,B 0,C 180,E1 -11424.401,E2 -11424.401} C_VEL
LIN {X 0,Y 395.896,Z 529.425,A -85,B 0,C 180,E1 -11425.928,E2 -11425.928} C_VEL
LIN {X 0,Y 395.867,Z 530.824,A -85,B 0,C 180,E1 -11426.947,E2 -11426.947} C_VEL
LIN {X 0,Y 395.86,Z 531.818,A -85,B 0,C 180,E1 -11427.965,E2 -11427.965} C_VEL
LIN {X 0,Y 395.779,Z 532.665,A -85,B 0,C 180,E1 -11430,E2 -11430} C_VEL
LIN {X 0,Y 395.797,Z 532.476,A -85,B 0,C 180,E1 -11431.018,E2 -11431.018} C_VEL
LIN {X 0,Y 395.86,Z 531.891,A -85,B 0,C 180,E1 -11432.035,E2 -11432.035} C_VEL
LIN {X 0,Y 395.886,Z 529.572,A -85,B 0,C 180,E1 -11434.072,E2 -11434.072} C_VEL
LIN {X 0,Y 396.148,Z 526.704,A -85,B 0,C 180,E1 -11435.6,E2 -11435.6} C_VEL
LIN {X 0,Y 396.328,Z 522.821,A -85,B 0,C 180,E1 -11437.131,E2 -11437.131} C_VEL
LIN {X 0,Y 396.688,Z 517.809,A -85,B 0,C 180,E1 -11438.661,E2 -11438.661} C_VEL
LIN {X 0,Y 397.26,Z 511.496,A -85,B 0,C 180,E1 -11440.19,E2 -11440.19} C_VEL
LIN {X 0,Y 397.963,Z 503.593,A -85,B 0,C 180,E1 -11441.718,E2 -11441.718} C_VEL
LIN {X 0,Y 398.874,Z 493.76,A -85,B 0,C 180,E1 -11443.242,E2 -11443.242} C_VEL
LIN {X 0,Y 399.708,Z 484.105,A -85,B 0,C 180,E1 -11444.437,E2 -11444.437} C_VEL
LIN {X 0,Y 400.436,Z 473.331,A -85,B 0,C 180,E1 -11445.514,E2 -11445.514} C_VEL
LIN {X 0,Y 400.156,Z 468.322,A -85,B 0,C 180,E1 -11445.967,E2 -11445.967} C_VEL
LIN {X 0,Y 398.953,Z 463.361,A -85,B 0,C 180,E1 -11446.411,E2 -11446.411} C_VEL
LIN {X 0,Y 395.351,Z 453.405,A -85,B 0,C 180,E1 -11447.24,E2 -11447.24} C_VEL
LIN {X 0,Y 393.288,Z 446.38,A -85,B 0,C 180,E1 -11447.722,E2 -11447.722} C_VEL
LIN {X 0,Y 390.339,Z 433.713,A -85,B 0,C 180,E1 -11448.387,E2 -11448.387} C_VEL
LIN {X 0,Y 389.09,Z 428.529,A -85,B 0,C 180,E1 -11448.632,E2 -11448.632} C_VEL
LIN {X 0,Y 389.177,Z 425.088,A -85,B 0,C 180,E1 -11451.172,E2 -11451.172} C_VEL
LIN {X 0,Y 389.379,Z 420.744,A -85,B 0,C 180,E1 -11454.528,E2 -11454.528} C_VEL
LIN {X 0,Y 389.593,Z 416.419,A -85,B 0,C 180,E1 -11457.971,E2 -11457.971} C_VEL
LIN {X 0,Y 389.824,Z 412.128,A -85,B 0,C 180,E1 -11461.523,E2 -11461.523} C_VEL
LIN {X 0,Y 389.949,Z 409.211,A -85,B 0,C 180,E1 -11463.998,E2 -11463.998} C_VEL
LIN {X 0,Y 389.969,Z 407.136,A -85,B 0,C 180,E1 -11465.807,E2 -11465.807} C_VEL
LIN {X 0,Y 390.091,Z 406.895,A -85,B 0,C 180,E1 -11469.092,E2 -11469.092} C_VEL
LIN {X 0,Y 390.047,Z 406.899,A -85,B 0,C 180,E1 -11472.374,E2 -11472.374} C_VEL
LIN {X 0,Y 390.048,Z 406.897,A -85,B 0,C 180,E1 -11475.355,E2 -11475.355} C_VEL
LIN {X 0,Y 390.033,Z 406.9,A -85,B 0,C 180,E1 -11478.187,E2 -11478.187} C_VEL
LIN {X 0,Y 390.094,Z 406.893,A -85,B 0,C 180,E1 -11480.908,E2 -11480.908} C_VEL
LIN {X 0,Y 390.088,Z 406.895,A -85,B 0,C 180,E1 -11484.793,E2 -11484.793} C_VEL
LIN {X 0,Y 390.027,Z 406.904,A -85,B 0,C 180,E1 -11488.496,E2 -11488.496} C_VEL
LIN {X 0,Y 390.12,Z 406.89,A -85,B 0,C 180,E1 -11492.07,E2 -11492.07} C_VEL
LIN {X 0,Y 390.082,Z 406.892,A -85,B 0,C 180,E1 -11495.519,E2 -11495.519} C_VEL
LIN {X 0,Y 390.059,Z 406.896,A -85,B 0,C 180,E1 -11498.878,E2 -11498.878} C_VEL
LIN {X 0,Y 390.13,Z 406.891,A -85,B 0,C 180,E1 -11502.167,E2 -11502.167} C_VEL
LIN {X 0,Y 390.147,Z 406.884,A -85,B 0,C 180,E1 -11505.393,E2 -11505.393} C_VEL
LIN {X 0,Y 390.151,Z 406.884,A -85,B 0,C 180,E1 -11508.571,E2 -11508.571} C_VEL
LIN {X 0,Y 390.347,Z 406.864,A -85,B 0,C 180,E1 -11511.993,E2 -11511.993} C_VEL
LIN {X 0,Y 390.229,Z 406.874,A -85,B 0,C 180,E1 -11514.833,E2 -11514.833} C_VEL
LIN {X 0,Y 390.421,Z 406.855,A -85,B 0,C 180,E1 -11517.937,E2 -11517.937} C_VEL
LIN {X 0,Y 390.551,Z 406.838,A -85,B 0,C 180,E1 -11520,E2 -11520} C_VEL
LIN {X 0,Y 390.313,Z 406.864,A -85,B 0,C 180,E1 -11523.096,E2 -11523.096} C_VEL
LIN {X 0,Y 390.333,Z 406.863,A -85,B 0,C 180,E1 -11526.202,E2 -11526.202} C_VEL
LIN {X 0,Y 390.318,Z 406.864,A -85,B 0,C 180,E1 -11528.282,E2 -11528.282} C_VEL
LIN {X 0,Y 390.181,Z 406.879,A -85,B 0,C 180,E1 -11532.483,E2 -11532.483} C_VEL
LIN {X 0,Y 390.143,Z 406.888,A -85,B 0,C 180,E1 -11535.677,E2 -11535.677} C_VEL
LIN {X 0,Y 390.109,Z 406.89,A -85,B 0,C 180,E1 -11538.922,E2 -11538.922} C_VEL
LIN {X 0,Y 390.042,Z 406.897,A -85,B 0,C 180,E1 -11542.234,E2 -11542.234} C_VEL
LIN {X 0,Y 390.121,Z 406.889,A -85,B 0,C 180,E1 -11545.743,E2 -11545.743} C_VEL
LIN {X 0,Y 390.061,Z 406.899,A -85,B 0,C 180,E1 -11549.109,E2 -11549.109} C_VEL
LIN {X 0,Y 390.045,Z 406.899,A -85,B 0,C 180,E1 -11552.721,E2 -11552.721} C_VEL
LIN {X 0,Y 390.06,Z 406.895,A -85,B 0,C 180,E1 -11555.826,E2 -11555.826} C_VEL
LIN {X 0,Y 390.074,Z 406.897,A -85,B 0,C 180,E1 -11559.219,E2 -11559.219} C_VEL
LIN {X 0,Y 390.044,Z 406.897,A -85,B 0,C 180,E1 -11562.374,E2 -11562.374} C_VEL
LIN {X 0,Y 390.049,Z 406.899,A -85,B 0,C 180,E1 -11565.355,E2 -11565.355} C_VEL
LIN {X 0,Y 390.073,Z 407.065,A -85,B 0,C 180,E1 -11568.319,E2 -11568.319} C_VEL
LIN {X 0,Y 391.003,Z 412.246,A -85,B 0,C 180,E1 -11571.675,E2 -11571.675} C_VEL
LIN {X 0,Y 391.383,Z 415.899,A -85,B 0,C 180,E1 -11573.907,E2 -11573.907} C_VEL
LIN {X 0,Y 391.211,Z 419.801,A -85,B 0,C 180,E1 -11576.158,E2 -11576.158} C_VEL
LIN {X 0,Y 390.725,Z 426.191,A -85,B 0,C 180,E1 -11579.699,E2 -11579.699} C_VEL
LIN {X 0,Y 390.185,Z 432.829,A -85,B 0,C 180,E1 -11583.237,E2 -11583.237} C_VEL
LIN {X 0,Y 389.768,Z 439.284,A -85,B 0,C 180,E1 -11586.629,E2 -11586.629} C_VEL
LIN {X 0,Y 389.451,Z 445.693,A -85,B 0,C 180,E1 -11589.948,E2 -11589.948} C_VEL
LIN {X 0,Y 389.28,Z 448.702,A -85,B 0,C 180,E1 -11591.429,E2 -11591.429} C_VEL
LIN {X 0,Y 391.853,Z 461.777,A -85,B 0,C 180,E1 -11591.978,E2 -11591.978} C_VEL
LIN {X 0,Y 393.57,Z 474.141,A -85,B 0,C 180,E1 -11592.671,E2 -11592.671} C_VEL
LIN {X 0,Y 394.176,Z 480.623,A -85,B 0,C 180,E1 -11593.105,E2 -11593.105} C_VEL
LIN {X 0,Y 393.391,Z 491.727,A -85,B 0,C 180,E1 -11593.924,E2 -11593.924} C_VEL
LIN {X 0,Y 392.427,Z 503.176,A -85,B 0,C 180,E1 -11595.002,E2 -11595.002} C_VEL
LIN {X 0,Y 391.557,Z 513.824,A -85,B 0,C 180,E1 -11596.273,E2 -11596.273} C_VEL
LIN {X 0,Y 390.79,Z 522.439,A -85,B 0,C 180,E1 -11597.537,E2 -11597.537} C_VEL
LIN {X 0,Y 389.931,Z 531.063,A -85,B 0,C 180,E1 -11599.091,E2 -11599.091} C_VEL
LIN {X 0,Y 389.41,Z 537.963,A -85,B 0,C 180,E1 -11600.652,E2 -11600.652} C_VEL
LIN {X 0,Y 389.043,Z 543.494,A -85,B 0,C 180,E1 -11602.213,E2 -11602.213} C_VEL
LIN {X 0,Y 388.775,Z 548.028,A -85,B 0,C 180,E1 -11603.855,E2 -11603.855} C_VEL
LIN {X 0,Y 388.746,Z 550.131,A -85,B 0,C 180,E1 -11604.814,E2 -11604.814} C_VEL
LIN {X 0,Y 388.703,Z 551.994,A -85,B 0,C 180,E1 -11605.852,E2 -11605.852} C_VEL
LIN {X 0,Y 388.662,Z 554.387,A -85,B 0,C 180,E1 -11607.927,E2 -11607.927} C_VEL
LIN {X 0,Y 388.703,Z 554.997,A -85,B 0,C 180,E1 -11608.964,E2 -11608.964} C_VEL
LIN {X 0,Y 388.707,Z 555.212,A -85,B 0,C 180,E1 -11610,E2 -11610} C_VEL
LIN {X 0,Y 388.703,Z 554.994,A -85,B 0,C 180,E1 -11611.036,E2 -11611.036} C_VEL
LIN {X 0,Y 388.662,Z 554.384,A -85,B 0,C 180,E1 -11612.072,E2 -11612.072} C_VEL
LIN {X 0,Y 388.703,Z 551.988,A -85,B 0,C 180,E1 -11614.147,E2 -11614.147} C_VEL
LIN {X 0,Y 388.731,Z 548.931,A -85,B 0,C 180,E1 -11615.76,E2 -11615.76} C_VEL
LIN {X 0,Y 388.941,Z 545.067,A -85,B 0,C 180,E1 -11617.267,E2 -11617.267} C_VEL
LIN {X 0,Y 389.356,Z 538.951,A -85,B 0,C 180,E1 -11619.087,E2 -11619.087} C_VEL
LIN {X 0,Y 389.865,Z 532.269,A -85,B 0,C 180,E1 -11620.648,E2 -11620.648} C_VEL
LIN {X 0,Y 390.649,Z 523.984,A -85,B 0,C 180,E1 -11622.204,E2 -11622.204} C_VEL
LIN {X 0,Y 391.399,Z 515.49,A -85,B 0,C 180,E1 -11623.499,E2 -11623.499} C_VEL
LIN {X 0,Y 392.256,Z 505.232,A -85,B 0,C 180,E1 -11624.765,E2 -11624.765} C_VEL
LIN {X 0,Y 393.169,Z 494.614,A -85,B 0,C 180,E1 -11625.819,E2 -11625.819} C_VEL
LIN {X 0,Y 393.977,Z 483.594,A -85,B 0,C 180,E1 -11626.69,E2 -11626.69} C_VEL
LIN {X 0,Y 394.087,Z 478.94,A -85,B 0,C 180,E1 -11627.004,E2 -11627.004} C_VEL
LIN {X 0,Y 392.55,Z 466.325,A -85,B 0,C 180,E1 -11627.78,E2 -11627.78} C_VEL
LIN {X 0,Y 390.192,Z 453.067,A -85,B 0,C 180,E1 -11628.398,E2 -11628.398} C_VEL
LIN {X 0,Y 389.273,Z 448.507,A -85,B 0,C 180,E1 -11628.588,E2 -11628.588} C_VEL
LIN {X 0,Y 389.621,Z 442.494,A -85,B 0,C 180,E1 -11631.702,E2 -11631.702} C_VEL
LIN {X 0,Y 389.976,Z 436.029,A -85,B 0,C 180,E1 -11635.056,E2 -11635.056} C_VEL
LIN {X 0,Y 390.374,Z 430.281,A -85,B 0,C 180,E1 -11638.096,E2 -11638.096} C_VEL
LIN {X 0,Y 390.783,Z 425.188,A -85,B 0,C 180,E1 -11640.834,E2 -11640.834} C_VEL
LIN {X 0,Y 391.285,Z 418.967,A -85,B 0,C 180,E1 -11644.287,E2 -11644.287} C_VEL
LIN {X 0,Y 391.325,Z 415.446,A -85,B 0,C 180,E1 -11646.346,E2 -11646.346} C_VEL
LIN {X 0,Y 390.863,Z 411.141,A -85,B 0,C 180,E1 -11649,E2 -11649} C_VEL
LIN {X 0,Y 390.053,Z 406.902,A -85,B 0,C 180,E1 -11651.81,E2 -11651.81} C_VEL
LIN {X 0,Y 390.047,Z 406.902,A -85,B 0,C 180,E1 -11655.355,E2 -11655.355} C_VEL
LIN {X 0,Y 390.032,Z 406.898,A -85,B 0,C 180,E1 -11658.187,E2 -11658.187} C_VEL
LIN {X 0,Y 390.093,Z 406.896,A -85,B 0,C 180,E1 -11660.908,E2 -11660.908} C_VEL
LIN {X 0,Y 390.087,Z 406.896,A -85,B 0,C 180,E1 -11664.793,E2 -11664.793} C_VEL
LIN {X 0,Y 390.025,Z 406.902,A -85,B 0,C 180,E1 -11668.496,E2 -11668.496} C_VEL
LIN {X 0,Y 390.118,Z 406.887,A -85,B 0,C 180,E1 -11672.07,E2 -11672.07} C_VEL
LIN {X 0,Y 390.08,Z 406.892,A -85,B 0,C 180,E1 -11675.519,E2 -11675.519} C_VEL
LIN {X 0,Y 390.057,Z 406.899,A -85,B 0,C 180,E1 -11678.878,E2 -11678.878} C_VEL
LIN {X 0,Y 390.13,Z 406.888,A -85,B 0,C 180,E1 -11682.167,E2 -11682.167} C_VEL
LIN {X 0,Y 390.149,Z 406.883,A -85,B 0,C 180,E1 -11685.393,E2 -11685.393} C_VEL
LIN {X 0,Y 390.161,Z 406.887,A -85,B 0,C 180,E1 -11688.572,E2 -11688.572} C_VEL
LIN {X 0,Y 390.346,Z 406.862,A -85,B 0,C 180,E1 -11691.993,E2 -11691.993} C_VEL
LIN {X 0,Y 390.228,Z 406.875,A -85,B 0,C 180,E1 -11694.834,E2 -11694.834} C_VEL
LIN {X 0,Y 390.42,Z 406.853,A -85,B 0,C 180,E1 -11697.937,E2 -11697.937} C_VEL
LIN {X 0,Y 390.552,Z 406.837,A -85,B 0,C 180,E1 -11700,E2 -11700} C_VEL
LIN {X 0,Y 390.311,Z 406.864,A -85,B 0,C 180,E1 -11703.097,E2 -11703.097} C_VEL
LIN {X 0,Y 390.311,Z 406.865,A -85,B 0,C 180,E1 -11706.65,E2 -11706.65} C_VEL
LIN {X 0,Y 390.212,Z 406.876,A -85,B 0,C 180,E1 -11709.329,E2 -11709.329} C_VEL
LIN {X 0,Y 390.18,Z 406.881,A -85,B 0,C 180,E1 -11712.483,E2 -11712.483} C_VEL
LIN {X 0,Y 390.142,Z 406.888,A -85,B 0,C 180,E1 -11715.677,E2 -11715.677} C_VEL
LIN {X 0,Y 390.106,Z 406.889,A -85,B 0,C 180,E1 -11718.922,E2 -11718.922} C_VEL
LIN {X 0,Y 390.041,Z 406.899,A -85,B 0,C 180,E1 -11722.234,E2 -11722.234} C_VEL
LIN {X 0,Y 390.12,Z 406.893,A -85,B 0,C 180,E1 -11725.743,E2 -11725.743} C_VEL
LIN {X 0,Y 390.06,Z 406.896,A -85,B 0,C 180,E1 -11729.11,E2 -11729.11} C_VEL
LIN {X 0,Y 390.044,Z 406.897,A -85,B 0,C 180,E1 -11732.722,E2 -11732.722} C_VEL
LIN {X 0,Y 390.059,Z 406.898,A -85,B 0,C 180,E1 -11735.826,E2 -11735.826} C_VEL
LIN {X 0,Y 390.074,Z 406.896,A -85,B 0,C 180,E1 -11739.219,E2 -11739.219} C_VEL
LIN {X 0,Y 390.044,Z 406.897,A -85,B 0,C 180,E1 -11742.374,E2 -11742.374} C_VEL
LIN {X 0,Y 390.048,Z 406.901,A -85,B 0,C 180,E1 -11745.355,E2 -11745.355} C_VEL
LIN {X 0,Y 390.034,Z 406.898,A -85,B 0,C 180,E1 -11748.187,E2 -11748.187} C_VEL
LIN {X 0,Y 390.09,Z 406.894,A -85,B 0,C 180,E1 -11750.908,E2 -11750.908} C_VEL
LIN {X 0,Y 389.932,Z 407.036,A -85,B 0,C 180,E1 -11754.2,E2 -11754.2} C_VEL
LIN {X 0,Y 389.876,Z 410.569,A -85,B 0,C 180,E1 -11757.263,E2 -11757.263} C_VEL
LIN {X 0,Y 389.666,Z 414.861,A -85,B 0,C 180,E1 -11760.858,E2 -11760.858} C_VEL
LIN {X 0,Y 389.454,Z 419.31,A -85,B 0,C 180,E1 -11764.461,E2 -11764.461} C_VEL
LIN {X 0,Y 389.242,Z 423.504,A -85,B 0,C 180,E1 -11767.718,E2 -11767.718} C_VEL
LIN {X 0,Y 389.106,Z 427.927,A -85,B 0,C 180,E1 -11771.028,E2 -11771.028} C_VEL
LIN {X 0,Y 389.093,Z 428.57,A -85,B 0,C 180,E1 -11771.498,E2 -11771.498} C_VEL
LIN {X 0,Y 392.31,Z 441.601,A -85,B 0,C 180,E1 -11772.11,E2 -11772.11} C_VEL
LIN {X 0,Y 394.718,Z 454.055,A -85,B 0,C 180,E1 -11772.868,E2 -11772.868} C_VEL
LIN {X 0,Y 394.291,Z 464.456,A -85,B 0,C 180,E1 -11773.563,E2 -11773.563} C_VEL
LIN {X 0,Y 393.485,Z 475.216,A -85,B 0,C 180,E1 -11774.46,E2 -11774.46} C_VEL
LIN {X 0,Y 392.733,Z 486.177,A -85,B 0,C 180,E1 -11775.623,E2 -11775.623} C_VEL
LIN {X 0,Y 391.839,Z 495.081,A -85,B 0,C 180,E1 -11776.781,E2 -11776.781} C_VEL
LIN {X 0,Y 391.07,Z 503.246,A -85,B 0,C 180,E1 -11778.073,E2 -11778.073} C_VEL
LIN {X 0,Y 390.317,Z 511.245,A -85,B 0,C 180,E1 -11779.627,E2 -11779.627} C_VEL
LIN {X 0,Y 389.684,Z 517.666,A -85,B 0,C 180,E1 -11781.182,E2 -11781.182} C_VEL
LIN {X 0,Y 389.313,Z 522.756,A -85,B 0,C 180,E1 -11782.74,E2 -11782.74} C_VEL
LIN {X 0,Y 389.085,Z 526.707,A -85,B 0,C 180,E1 -11784.299,E2 -11784.299} C_VEL
LIN {X 0,Y 388.822,Z 529.63,A -85,B 0,C 180,E1 -11785.854,E2 -11785.854} C_VEL
LIN {X 0,Y 388.772,Z 531.028,A -85,B 0,C 180,E1 -11786.891,E2 -11786.891} C_VEL
LIN {X 0,Y 388.763,Z 532.022,A -85,B 0,C 180,E1 -11787.928,E2 -11787.928} C_VEL
LIN {X 0,Y 388.708,Z 532.868,A -85,B 0,C 180,E1 -11790,E2 -11790} C_VEL
LIN {X 0,Y 388.729,Z 532.679,A -85,B 0,C 180,E1 -11791.036,E2 -11791.036} C_VEL
LIN {X 0,Y 388.762,Z 532.094,A -85,B 0,C 180,E1 -11792.072,E2 -11792.072} C_VEL
LIN {X 0,Y 388.813,Z 529.775,A -85,B 0,C 180,E1 -11794.146,E2 -11794.146} C_VEL
LIN {X 0,Y 389.079,Z 526.907,A -85,B 0,C 180,E1 -11795.702,E2 -11795.702} C_VEL
LIN {X 0,Y 389.28,Z 523.024,A -85,B 0,C 180,E1 -11797.26,E2 -11797.26} C_VEL
LIN {X 0,Y 389.673,Z 518.011,A -85,B 0,C 180,E1 -11798.819,E2 -11798.819} C_VEL
LIN {X 0,Y 390.27,Z 511.698,A -85,B 0,C 180,E1 -11800.375,E2 -11800.375} C_VEL
LIN {X 0,Y 391.013,Z 503.794,A -85,B 0,C 180,E1 -11801.929,E2 -11801.929} C_VEL
LIN {X 0,Y 391.959,Z 493.961,A -85,B 0,C 180,E1 -11803.48,E2 -11803.48} C_VEL
LIN {X 0,Y 392.82,Z 484.626,A -85,B 0,C 180,E1 -11804.659,E2 -11804.659} C_VEL
LIN {X 0,Y 393.57,Z 473.939,A -85,B 0,C 180,E1 -11805.754,E2 -11805.754} C_VEL
LIN {X 0,Y 394.439,Z 462.597,A -85,B 0,C 180,E1 -11806.669,E2 -11806.669} C_VEL
LIN {X 0,Y 394.834,Z 454.837,A -85,B 0,C 180,E1 -11807.179,E2 -11807.179} C_VEL
LIN {X 0,Y 393.288,Z 446.38,A -85,B 0,C 180,E1 -11807.722,E2 -11807.722} C_VEL
LIN {X 0,Y 391.879,Z 443.015,A -85,B 0,C 180,E1 -11807.954,E2 -11807.954} C_VEL
LIN {X 0,Y 387.893,Z 438.276,A -85,B 0,C 180,E1 -11808.351,E2 -11808.351} C_VEL
LIN {X 0,Y 383.824,Z 433.482,A -85,B 0,C 180,E1 -11808.723,E2 -11808.723} C_VEL
LIN {X 0,Y 382.265,Z 430.023,A -85,B 0,C 180,E1 -11808.909,E2 -11808.909} C_VEL
LIN {X 0,Y 382.036,Z 428.725,A -85,B 0,C 180,E1 -11808.989,E2 -11808.989} C_VEL
LIN {X 0,Y 382.12,Z 425.278,A -85,B 0,C 180,E1 -11811.583,E2 -11811.583} C_VEL
LIN {X 0,Y 382.259,Z 422.369,A -85,B 0,C 180,E1 -11813.859,E2 -11813.859} C_VEL
LIN {X 0,Y 382.444,Z 419.459,A -85,B 0,C 180,E1 -11816.17,E2 -11816.17} C_VEL
LIN {X 0,Y 382.639,Z 415.146,A -85,B 0,C 180,E1 -11819.73,E2 -11819.73} C_VEL
LIN {X 0,Y 382.821,Z 412.008,A -85,B 0,C 180,E1 -11822.382,E2 -11822.382} C_VEL
LIN {X 0,Y 382.932,Z 409.391,A -85,B 0,C 180,E1 -11824.677,E2 -11824.677} C_VEL
LIN {X 0,Y 382.929,Z 407.788,A -85,B 0,C 180,E1 -11826.143,E2 -11826.143} C_VEL
LIN {X 0,Y 383.017,Z 407.772,A -85,B 0,C 180,E1 -11829.586,E2 -11829.586} C_VEL
LIN {X 0,Y 383.008,Z 407.778,A -85,B 0,C 180,E1 -11832.779,E2 -11832.779} C_VEL
LIN {X 0,Y 383,Z 407.774,A -85,B 0,C 180,E1 -11835.789,E2 -11835.789} C_VEL
LIN {X 0,Y 382.991,Z 407.78,A -85,B 0,C 180,E1 -11838.796,E2 -11838.796} C_VEL
LIN {X 0,Y 383.004,Z 407.775,A -85,B 0,C 180,E1 -11842.096,E2 -11842.096} C_VEL
LIN {X 0,Y 383.021,Z 407.772,A -85,B 0,C 180,E1 -11845.332,E2 -11845.332} C_VEL
LIN {X 0,Y 382.986,Z 407.777,A -85,B 0,C 180,E1 -11849.081,E2 -11849.081} C_VEL
LIN {X 0,Y 383.059,Z 407.769,A -85,B 0,C 180,E1 -11852.698,E2 -11852.698} C_VEL
LIN {X 0,Y 383.054,Z 407.767,A -85,B 0,C 180,E1 -11855.04,E2 -11855.04} C_VEL
LIN {X 0,Y 382.996,Z 407.779,A -85,B 0,C 180,E1 -11858.469,E2 -11858.469} C_VEL
LIN {X 0,Y 383.065,Z 407.769,A -85,B 0,C 180,E1 -11861.826,E2 -11861.826} C_VEL
LIN {X 0,Y 383.113,Z 407.76,A -85,B 0,C 180,E1 -11865.118,E2 -11865.118} C_VEL
LIN {X 0,Y 383.101,Z 407.764,A -85,B 0,C 180,E1 -11868.358,E2 -11868.358} C_VEL
LIN {X 0,Y 383.307,Z 407.741,A -85,B 0,C 180,E1 -11871.933,E2 -11871.933} C_VEL
LIN {X 0,Y 383.201,Z 407.749,A -85,B 0,C 180,E1 -11874.738,E2 -11874.738} C_VEL
LIN {X 0,Y 383.388,Z 407.731,A -85,B 0,C 180,E1 -11877.899,E2 -11877.899} C_VEL
LIN {X 0,Y 383.521,Z 407.713,A -85,B 0,C 180,E1 -11880,E2 -11880} C_VEL
LIN {X 0,Y 383.249,Z 407.744,A -85,B 0,C 180,E1 -11883.154,E2 -11883.154} C_VEL
LIN {X 0,Y 383.29,Z 407.739,A -85,B 0,C 180,E1 -11886.316,E2 -11886.316} C_VEL
LIN {X 0,Y 383.264,Z 407.742,A -85,B 0,C 180,E1 -11888.436,E2 -11888.436} C_VEL
LIN {X 0,Y 383.111,Z 407.766,A -85,B 0,C 180,E1 -11891.642,E2 -11891.642} C_VEL
LIN {X 0,Y 383.115,Z 407.76,A -85,B 0,C 180,E1 -11894.882,E2 -11894.882} C_VEL
LIN {X 0,Y 383.066,Z 407.766,A -85,B 0,C 180,E1 -11898.173,E2 -11898.173} C_VEL
LIN {X 0,Y 382.996,Z 407.78,A -85,B 0,C 180,E1 -11901.531,E2 -11901.531} C_VEL
LIN {X 0,Y 383.054,Z 407.77,A -85,B 0,C 180,E1 -11904.96,E2 -11904.96} C_VEL
LIN {X 0,Y 383.032,Z 407.769,A -85,B 0,C 180,E1 -11908.27,E2 -11908.27} C_VEL
LIN {X 0,Y 383.012,Z 407.772,A -85,B 0,C 180,E1 -11912.15,E2 -11912.15} C_VEL
LIN {X 0,Y 383.021,Z 407.774,A -85,B 0,C 180,E1 -11914.668,E2 -11914.668} C_VEL
LIN {X 0,Y 383.004,Z 407.774,A -85,B 0,C 180,E1 -11917.904,E2 -11917.904} C_VEL
LIN {X 0,Y 382.986,Z 407.778,A -85,B 0,C 180,E1 -11921.347,E2 -11921.347} C_VEL
LIN {X 0,Y 382.999,Z 407.78,A -85,B 0,C 180,E1 -11924.303,E2 -11924.303} C_VEL
LIN {X 0,Y 383.012,Z 407.841,A -85,B 0,C 180,E1 -11927.952,E2 -11927.952} C_VEL
LIN {X 0,Y 383.976,Z 413.205,A -85,B 0,C 180,E1 -11931.515,E2 -11931.515} C_VEL
LIN {X 0,Y 384.382,Z 417.517,A -85,B 0,C 180,E1 -11934.191,E2 -11934.191} C_VEL
LIN {X 0,Y 384.119,Z 421.842,A -85,B 0,C 180,E1 -11936.709,E2 -11936.709} C_VEL
LIN {X 0,Y 383.579,Z 428.331,A -85,B 0,C 180,E1 -11940.35,E2 -11940.35} C_VEL
LIN {X 0,Y 383.017,Z 435.121,A -85,B 0,C 180,E1 -11944.041,E2 -11944.041} C_VEL
LIN {X 0,Y 382.591,Z 442.326,A -85,B 0,C 180,E1 -11947.878,E2 -11947.878} C_VEL
LIN {X 0,Y 382.223,Z 448.505,A -85,B 0,C 180,E1 -11951.073,E2 -11951.073} C_VEL
LIN {X 0,Y 384.805,Z 461.459,A -85,B 0,C 180,E1 -11951.631,E2 -11951.631} C_VEL
LIN {X 0,Y 386.516,Z 473.149,A -85,B 0,C 180,E1 -11952.297,E2 -11952.297} C_VEL
LIN {X 0,Y 387.311,Z 482.177,A -85,B 0,C 180,E1 -11952.916,E2 -11952.916} C_VEL
LIN {X 0,Y 386.347,Z 494.492,A -85,B 0,C 180,E1 -11953.894,E2 -11953.894} C_VEL
LIN {X 0,Y 385.282,Z 506.035,A -85,B 0,C 180,E1 -11955.069,E2 -11955.069} C_VEL
LIN {X 0,Y 384.471,Z 515.338,A -85,B 0,C 180,E1 -11956.253,E2 -11956.253} C_VEL
LIN {X 0,Y 383.666,Z 523.82,A -85,B 0,C 180,E1 -11957.57,E2 -11957.57} C_VEL
LIN {X 0,Y 382.84,Z 532.097,A -85,B 0,C 180,E1 -11959.154,E2 -11959.154} C_VEL
LIN {X 0,Y 382.293,Z 538.773,A -85,B 0,C 180,E1 -11960.743,E2 -11960.743} C_VEL
LIN {X 0,Y 381.871,Z 544.883,A -85,B 0,C 180,E1 -11962.598,E2 -11962.598} C_VEL
LIN {X 0,Y 381.672,Z 548.209,A -85,B 0,C 180,E1 -11963.904,E2 -11963.904} C_VEL
LIN {X 0,Y 381.628,Z 551.791,A -85,B 0,C 180,E1 -11965.775,E2 -11965.775} C_VEL
LIN {X 0,Y 381.56,Z 554.183,A -85,B 0,C 180,E1 -11967.889,E2 -11967.889} C_VEL
LIN {X 0,Y 381.617,Z 554.793,A -85,B 0,C 180,E1 -11968.945,E2 -11968.945} C_VEL
LIN {X 0,Y 381.639,Z 555.009,A -85,B 0,C 180,E1 -11970,E2 -11970} C_VEL
LIN {X 0,Y 381.617,Z 554.791,A -85,B 0,C 180,E1 -11971.055,E2 -11971.055} C_VEL
LIN {X 0,Y 381.548,Z 553.181,A -85,B 0,C 180,E1 -11973.168,E2 -11973.168} C_VEL
LIN {X 0,Y 381.628,Z 551.783,A -85,B 0,C 180,E1 -11974.224,E2 -11974.224} C_VEL
LIN {X 0,Y 381.672,Z 548.193,A -85,B 0,C 180,E1 -11976.096,E2 -11976.096} C_VEL
LIN {X 0,Y 381.989,Z 543.267,A -85,B 0,C 180,E1 -11977.931,E2 -11977.931} C_VEL
LIN {X 0,Y 382.388,Z 537.732,A -85,B 0,C 180,E1 -11979.521,E2 -11979.521} C_VEL
LIN {X 0,Y 382.93,Z 530.824,A -85,B 0,C 180,E1 -11981.111,E2 -11981.111} C_VEL
LIN {X 0,Y 383.847,Z 522.188,A -85,B 0,C 180,E1 -11982.692,E2 -11982.692} C_VEL
LIN {X 0,Y 384.795,Z 512.113,A -85,B 0,C 180,E1 -11984.172,E2 -11984.172} C_VEL
LIN {X 0,Y 385.566,Z 502.429,A -85,B 0,C 180,E1 -11985.325,E2 -11985.325} C_VEL
LIN {X 0,Y 386.555,Z 491.431,A -85,B 0,C 180,E1 -11986.368,E2 -11986.368} C_VEL
LIN {X 0,Y 387.278,Z 480.569,A -85,B 0,C 180,E1 -11987.187,E2 -11987.187} C_VEL
LIN {X 0,Y 385.879,Z 468.639,A -85,B 0,C 180,E1 -11987.969,E2 -11987.969} C_VEL
LIN {X 0,Y 383.851,Z 456.508,A -85,B 0,C 180,E1 -11988.595,E2 -11988.595} C_VEL
LIN {X 0,Y 382.219,Z 448.32,A -85,B 0,C 180,E1 -11988.944,E2 -11988.944} C_VEL
LIN {X 0,Y 382.59,Z 442.305,A -85,B 0,C 180,E1 -11992.122,E2 -11992.122} C_VEL
LIN {X 0,Y 383.017,Z 435.092,A -85,B 0,C 180,E1 -11995.959,E2 -11995.959} C_VEL
LIN {X 0,Y 383.619,Z 428.291,A -85,B 0,C 180,E1 -11999.646,E2 -11999.646} C_VEL
LIN {X 0,Y 384.117,Z 421.775,A -85,B 0,C 180,E1 -12003.291,E2 -12003.291} C_VEL
LIN {X 0,Y 384.359,Z 417.465,A -85,B 0,C 180,E1 -12005.811,E2 -12005.811} C_VEL
LIN {X 0,Y 384.061,Z 413.76,A -85,B 0,C 180,E1 -12008.106,E2 -12008.106} C_VEL
LIN {X 0,Y 383.221,Z 408.881,A -85,B 0,C 180,E1 -12011.316,E2 -12011.316} C_VEL
LIN {X 0,Y 383.025,Z 407.777,A -85,B 0,C 180,E1 -12012.223,E2 -12012.223} C_VEL
LIN {X 0,Y 382.999,Z 407.78,A -85,B 0,C 180,E1 -12015.789,E2 -12015.789} C_VEL
LIN {X 0,Y 382.989,Z 407.779,A -85,B 0,C 180,E1 -12018.796,E2 -12018.796} C_VEL
LIN {X 0,Y 383.003,Z 407.774,A -85,B 0,C 180,E1 -12022.096,E2 -12022.096} C_VEL
LIN {X 0,Y 383.019,Z 407.774,A -85,B 0,C 180,E1 -12025.332,E2 -12025.332} C_VEL
LIN {X 0,Y 382.984,Z 407.779,A -85,B 0,C 180,E1 -12029.081,E2 -12029.081} C_VEL
LIN {X 0,Y 383.058,Z 407.772,A -85,B 0,C 180,E1 -12032.698,E2 -12032.698} C_VEL
LIN {X 0,Y 383.053,Z 407.771,A -85,B 0,C 180,E1 -12035.04,E2 -12035.04} C_VEL
LIN {X 0,Y 382.994,Z 407.78,A -85,B 0,C 180,E1 -12038.469,E2 -12038.469} C_VEL
LIN {X 0,Y 383.064,Z 407.766,A -85,B 0,C 180,E1 -12041.826,E2 -12041.826} C_VEL
LIN {X 0,Y 383.114,Z 407.76,A -85,B 0,C 180,E1 -12045.118,E2 -12045.118} C_VEL
LIN {X 0,Y 383.11,Z 407.766,A -85,B 0,C 180,E1 -12048.358,E2 -12048.358} C_VEL
LIN {X 0,Y 383.305,Z 407.738,A -85,B 0,C 180,E1 -12051.933,E2 -12051.933} C_VEL
LIN {X 0,Y 383.2,Z 407.751,A -85,B 0,C 180,E1 -12054.739,E2 -12054.739} C_VEL
LIN {X 0,Y 383.387,Z 407.728,A -85,B 0,C 180,E1 -12057.899,E2 -12057.899} C_VEL
LIN {X 0,Y 383.522,Z 407.713,A -85,B 0,C 180,E1 -12060,E2 -12060} C_VEL
LIN {X 0,Y 383.248,Z 407.743,A -85,B 0,C 180,E1 -12063.154,E2 -12063.154} C_VEL
LIN {X 0,Y 383.271,Z 407.742,A -85,B 0,C 180,E1 -12066.645,E2 -12066.645} C_VEL
LIN {X 0,Y 383.262,Z 407.744,A -85,B 0,C 180,E1 -12068.436,E2 -12068.436} C_VEL
LIN {X 0,Y 383.109,Z 407.763,A -85,B 0,C 180,E1 -12071.642,E2 -12071.642} C_VEL
LIN {X 0,Y 383.114,Z 407.76,A -85,B 0,C 180,E1 -12074.882,E2 -12074.882} C_VEL
LIN {X 0,Y 383.064,Z 407.77,A -85,B 0,C 180,E1 -12078.174,E2 -12078.174} C_VEL
LIN {X 0,Y 382.995,Z 407.778,A -85,B 0,C 180,E1 -12081.531,E2 -12081.531} C_VEL
LIN {X 0,Y 383.053,Z 407.767,A -85,B 0,C 180,E1 -12084.96,E2 -12084.96} C_VEL
LIN {X 0,Y 383.031,Z 407.771,A -85,B 0,C 180,E1 -12088.27,E2 -12088.27} C_VEL
LIN {X 0,Y 383.011,Z 407.774,A -85,B 0,C 180,E1 -12092.15,E2 -12092.15} C_VEL
LIN {X 0,Y 383.02,Z 407.772,A -85,B 0,C 180,E1 -12094.668,E2 -12094.668} C_VEL
LIN {X 0,Y 383.004,Z 407.775,A -85,B 0,C 180,E1 -12097.904,E2 -12097.904} C_VEL
LIN {X 0,Y 382.987,Z 407.781,A -85,B 0,C 180,E1 -12101.347,E2 -12101.347} C_VEL
LIN {X 0,Y 382.999,Z 407.774,A -85,B 0,C 180,E1 -12104.304,E2 -12104.304} C_VEL
LIN {X 0,Y 383.011,Z 407.778,A -85,B 0,C 180,E1 -12107.24,E2 -12107.24} C_VEL
LIN {X 0,Y 383.016,Z 407.772,A -85,B 0,C 180,E1 -12110.414,E2 -12110.414} C_VEL
LIN {X 0,Y 382.969,Z 407.781,A -85,B 0,C 180,E1 -12112.728,E2 -12112.728} C_VEL
LIN {X 0,Y 382.897,Z 407.821,A -85,B 0,C 180,E1 -12114.031,E2 -12114.031} C_VEL
LIN {X 0,Y 382.857,Z 410.709,A -85,B 0,C 180,E1 -12116.585,E2 -12116.585} C_VEL
LIN {X 0,Y 382.704,Z 414.311,A -85,B 0,C 180,E1 -12119.668,E2 -12119.668} C_VEL
LIN {X 0,Y 382.486,Z 417.877,A -85,B 0,C 180,E1 -12122.654,E2 -12122.654} C_VEL
LIN {X 0,Y 382.341,Z 420.78,A -85,B 0,C 180,E1 -12124.99,E2 -12124.99} C_VEL
LIN {X 0,Y 382.224,Z 423.689,A -85,B 0,C 180,E1 -12127.286,E2 -12127.286} C_VEL
LIN {X 0,Y 382.071,Z 428.124,A -85,B 0,C 180,E1 -12130.664,E2 -12130.664} C_VEL
LIN {X 0,Y 382.064,Z 428.865,A -85,B 0,C 180,E1 -12131.147,E2 -12131.147} C_VEL
LIN {X 0,Y 385.372,Z 442.001,A -85,B 0,C 180,E1 -12131.785,E2 -12131.785} C_VEL
LIN {X 0,Y 387.837,Z 454.839,A -85,B 0,C 180,E1 -12132.589,E2 -12132.589} C_VEL
LIN {X 0,Y 387.794,Z 460.401,A -85,B 0,C 180,E1 -12132.958,E2 -12132.958} C_VEL
LIN {X 0,Y 386.98,Z 471.143,A -85,B 0,C 180,E1 -12133.786,E2 -12133.786} C_VEL
LIN {X 0,Y 386.23,Z 482.021,A -85,B 0,C 180,E1 -12134.861,E2 -12134.861} C_VEL
LIN {X 0,Y 385.369,Z 491.533,A -85,B 0,C 180,E1 -12136.017,E2 -12136.017} C_VEL
LIN {X 0,Y 384.388,Z 500.377,A -85,B 0,C 180,E1 -12137.326,E2 -12137.326} C_VEL
LIN {X 0,Y 383.568,Z 508.999,A -85,B 0,C 180,E1 -12138.908,E2 -12138.908} C_VEL
LIN {X 0,Y 382.889,Z 515.872,A -85,B 0,C 180,E1 -12140.491,E2 -12140.491} C_VEL
LIN {X 0,Y 382.346,Z 521.375,A -85,B 0,C 180,E1 -12142.076,E2 -12142.076} C_VEL
LIN {X 0,Y 382.104,Z 525.689,A -85,B 0,C 180,E1 -12143.664,E2 -12143.664} C_VEL
LIN {X 0,Y 381.955,Z 527.973,A -85,B 0,C 180,E1 -12144.721,E2 -12144.721} C_VEL
LIN {X 0,Y 381.751,Z 529.834,A -85,B 0,C 180,E1 -12145.777,E2 -12145.777} C_VEL
LIN {X 0,Y 381.678,Z 531.233,A -85,B 0,C 180,E1 -12146.833,E2 -12146.833} C_VEL
LIN {X 0,Y 381.666,Z 532.227,A -85,B 0,C 180,E1 -12147.89,E2 -12147.89} C_VEL
LIN {X 0,Y 381.64,Z 533.072,A -85,B 0,C 180,E1 -12150,E2 -12150} C_VEL
LIN {X 0,Y 381.644,Z 532.882,A -85,B 0,C 180,E1 -12151.055,E2 -12151.055} C_VEL
LIN {X 0,Y 381.665,Z 532.298,A -85,B 0,C 180,E1 -12152.111,E2 -12152.111} C_VEL
LIN {X 0,Y 381.743,Z 529.978,A -85,B 0,C 180,E1 -12154.223,E2 -12154.223} C_VEL
LIN {X 0,Y 382.012,Z 527.11,A -85,B 0,C 180,E1 -12155.808,E2 -12155.808} C_VEL
LIN {X 0,Y 382.242,Z 523.227,A -85,B 0,C 180,E1 -12157.395,E2 -12157.395} C_VEL
LIN {X 0,Y 382.647,Z 518.214,A -85,B 0,C 180,E1 -12158.982,E2 -12158.982} C_VEL
LIN {X 0,Y 383.273,Z 511.9,A -85,B 0,C 180,E1 -12160.566,E2 -12160.566} C_VEL
LIN {X 0,Y 384.061,Z 503.996,A -85,B 0,C 180,E1 -12162.148,E2 -12162.148} C_VEL
LIN {X 0,Y 385.059,Z 494.162,A -85,B 0,C 180,E1 -12163.726,E2 -12163.726} C_VEL
LIN {X 0,Y 386.011,Z 483.997,A -85,B 0,C 180,E1 -12165.019,E2 -12165.019} C_VEL
LIN {X 0,Y 386.791,Z 473.617,A -85,B 0,C 180,E1 -12166.087,E2 -12166.087} C_VEL
LIN {X 0,Y 387.764,Z 461.523,A -85,B 0,C 180,E1 -12167.063,E2 -12167.063} C_VEL
LIN {X 0,Y 387.927,Z 455.513,A -85,B 0,C 180,E1 -12167.466,E2 -12167.466} C_VEL
LIN {X 0,Y 386.018,Z 445.311,A -85,B 0,C 180,E1 -12168.133,E2 -12168.133} C_VEL
LIN {X 0,Y 382.907,Z 432.393,A -85,B 0,C 180,E1 -12168.803,E2 -12168.803} C_VEL
LIN {X 0,Y 382.265,Z 430.023,A -85,B 0,C 180,E1 -12168.909,E2 -12168.909} C_VEL
LIN {X 0,Y 381.65,Z 428.864,A -85,B 0,C 180,E1 -12169.069,E2 -12169.069} C_VEL
LIN {X 0,Y 378.773,Z 427.457,A -85,B 0,C 180,E1 -12170.191,E2 -12170.191} C_VEL
LIN {X 0,Y 376.297,Z 426.064,A -85,B 0,C 180,E1 -12171.76,E2 -12171.76} C_VEL
LIN {X 0,Y 375.209,Z 423.637,A -85,B 0,C 180,E1 -12173.464,E2 -12173.464} C_VEL
LIN {X 0,Y 375.405,Z 419.635,A -85,B 0,C 180,E1 -12176.699,E2 -12176.699} C_VEL
LIN {X 0,Y 375.635,Z 415.287,A -85,B 0,C 180,E1 -12180.342,E2 -12180.342} C_VEL
LIN {X 0,Y 375.866,Z 410.987,A -85,B 0,C 180,E1 -12184.121,E2 -12184.121} C_VEL
LIN {X 0,Y 375.904,Z 408.663,A -85,B 0,C 180,E1 -12186.492,E2 -12186.492} C_VEL
LIN {X 0,Y 375.991,Z 408.647,A -85,B 0,C 180,E1 -12189.971,E2 -12189.971} C_VEL
LIN {X 0,Y 375.933,Z 408.654,A -85,B 0,C 180,E1 -12193.766,E2 -12193.766} C_VEL
LIN {X 0,Y 375.937,Z 408.659,A -85,B 0,C 180,E1 -12196.81,E2 -12196.81} C_VEL
LIN {X 0,Y 375.966,Z 408.655,A -85,B 0,C 180,E1 -12200.538,E2 -12200.538} C_VEL
LIN {X 0,Y 375.967,Z 408.65,A -85,B 0,C 180,E1 -12203.495,E2 -12203.495} C_VEL
LIN {X 0,Y 375.962,Z 408.651,A -85,B 0,C 180,E1 -12205.889,E2 -12205.889} C_VEL
LIN {X 0,Y 375.967,Z 408.65,A -85,B 0,C 180,E1 -12209.687,E2 -12209.687} C_VEL
LIN {X 0,Y 376.022,Z 408.643,A -85,B 0,C 180,E1 -12213.348,E2 -12213.348} C_VEL
LIN {X 0,Y 375.999,Z 408.647,A -85,B 0,C 180,E1 -12216.888,E2 -12216.888} C_VEL
LIN {X 0,Y 376.001,Z 408.651,A -85,B 0,C 180,E1 -12220.339,E2 -12220.339} C_VEL
LIN {X 0,Y 376.032,Z 408.644,A -85,B 0,C 180,E1 -12223.719,E2 -12223.719} C_VEL
LIN {X 0,Y 376.106,Z 408.632,A -85,B 0,C 180,E1 -12227.042,E2 -12227.042} C_VEL
LIN {X 0,Y 376.122,Z 408.634,A -85,B 0,C 180,E1 -12230.319,E2 -12230.319} C_VEL
LIN {X 0,Y 376.233,Z 408.618,A -85,B 0,C 180,E1 -12232.486,E2 -12232.486} C_VEL
LIN {X 0,Y 376.174,Z 408.625,A -85,B 0,C 180,E1 -12234.64,E2 -12234.64} C_VEL
LIN {X 0,Y 376.354,Z 408.607,A -85,B 0,C 180,E1 -12237.86,E2 -12237.86} C_VEL
LIN {X 0,Y 376.49,Z 408.589,A -85,B 0,C 180,E1 -12240,E2 -12240} C_VEL
LIN {X 0,Y 376.188,Z 408.623,A -85,B 0,C 180,E1 -12243.213,E2 -12243.213} C_VEL
LIN {X 0,Y 376.25,Z 408.615,A -85,B 0,C 180,E1 -12246.435,E2 -12246.435} C_VEL
LIN {X 0,Y 376.209,Z 408.62,A -85,B 0,C 180,E1 -12248.595,E2 -12248.595} C_VEL
LIN {X 0,Y 376.062,Z 408.641,A -85,B 0,C 180,E1 -12251.863,E2 -12251.863} C_VEL
LIN {X 0,Y 376.063,Z 408.64,A -85,B 0,C 180,E1 -12255.167,E2 -12255.167} C_VEL
LIN {X 0,Y 376.012,Z 408.644,A -85,B 0,C 180,E1 -12258.527,E2 -12258.527} C_VEL
LIN {X 0,Y 375.965,Z 408.651,A -85,B 0,C 180,E1 -12261.954,E2 -12261.954} C_VEL
LIN {X 0,Y 376.009,Z 408.649,A -85,B 0,C 180,E1 -12265.461,E2 -12265.461} C_VEL
LIN {X 0,Y 375.963,Z 408.655,A -85,B 0,C 180,E1 -12269.08,E2 -12269.08} C_VEL
LIN {X 0,Y 375.951,Z 408.655,A -85,B 0,C 180,E1 -12272.828,E2 -12272.828} C_VEL
LIN {X 0,Y 375.961,Z 408.654,A -85,B 0,C 180,E1 -12275.415,E2 -12275.415} C_VEL
LIN {X 0,Y 375.978,Z 408.649,A -85,B 0,C 180,E1 -12278.271,E2 -12278.271} C_VEL
LIN {X 0,Y 375.936,Z 408.654,A -85,B 0,C 180,E1 -12281.601,E2 -12281.601} C_VEL
LIN {X 0,Y 375.931,Z 408.658,A -85,B 0,C 180,E1 -12285.268,E2 -12285.268} C_VEL
LIN {X 0,Y 376.006,Z 408.792,A -85,B 0,C 180,E1 -12287.71,E2 -12287.71} C_VEL
LIN {X 0,Y 377.002,Z 414.438,A -85,B 0,C 180,E1 -12291.532,E2 -12291.532} C_VEL
LIN {X 0,Y 377.375,Z 418.454,A -85,B 0,C 180,E1 -12294.081,E2 -12294.081} C_VEL
LIN {X 0,Y 377.201,Z 421.694,A -85,B 0,C 180,E1 -12296.016,E2 -12296.016} C_VEL
LIN {X 0,Y 376.605,Z 428.169,A -85,B 0,C 180,E1 -12299.744,E2 -12299.744} C_VEL
LIN {X 0,Y 376.133,Z 433.57,A -85,B 0,C 180,E1 -12302.756,E2 -12302.756} C_VEL
LIN {X 0,Y 375.657,Z 440.308,A -85,B 0,C 180,E1 -12306.451,E2 -12306.451} C_VEL
LIN {X 0,Y 375.352,Z 445.783,A -85,B 0,C 180,E1 -12309.421,E2 -12309.421} C_VEL
LIN {X 0,Y 375.215,Z 448.309,A -85,B 0,C 180,E1 -12310.706,E2 -12310.706} C_VEL
LIN {X 0,Y 377.839,Z 461.552,A -85,B 0,C 180,E1 -12311.294,E2 -12311.294} C_VEL
LIN {X 0,Y 379.615,Z 473.567,A -85,B 0,C 180,E1 -12312.002,E2 -12312.002} C_VEL
LIN {X 0,Y 380.401,Z 483.427,A -85,B 0,C 180,E1 -12312.706,E2 -12312.706} C_VEL
LIN {X 0,Y 379.39,Z 495.721,A -85,B 0,C 180,E1 -12313.729,E2 -12313.729} C_VEL
LIN {X 0,Y 378.421,Z 505.835,A -85,B 0,C 180,E1 -12314.792,E2 -12314.792} C_VEL
LIN {X 0,Y 377.54,Z 515.136,A -85,B 0,C 180,E1 -12315.995,E2 -12315.995} C_VEL
LIN {X 0,Y 376.71,Z 523.617,A -85,B 0,C 180,E1 -12317.337,E2 -12317.337} C_VEL
LIN {X 0,Y 375.814,Z 531.893,A -85,B 0,C 180,E1 -12318.949,E2 -12318.949} C_VEL
LIN {X 0,Y 375.249,Z 538.569,A -85,B 0,C 180,E1 -12320.568,E2 -12320.568} C_VEL
LIN {X 0,Y 374.808,Z 544.679,A -85,B 0,C 180,E1 -12322.458,E2 -12322.458} C_VEL
LIN {X 0,Y 374.568,Z 548.39,A -85,B 0,C 180,E1 -12323.954,E2 -12323.954} C_VEL
LIN {X 0,Y 374.554,Z 551.587,A -85,B 0,C 180,E1 -12325.696,E2 -12325.696} C_VEL
LIN {X 0,Y 374.46,Z 553.979,A -85,B 0,C 180,E1 -12327.849,E2 -12327.849} C_VEL
LIN {X 0,Y 374.517,Z 554.589,A -85,B 0,C 180,E1 -12328.925,E2 -12328.925} C_VEL
LIN {X 0,Y 374.554,Z 554.806,A -85,B 0,C 180,E1 -12330,E2 -12330} C_VEL
LIN {X 0,Y 374.517,Z 554.586,A -85,B 0,C 180,E1 -12331.075,E2 -12331.075} C_VEL
LIN {X 0,Y 374.463,Z 552.977,A -85,B 0,C 180,E1 -12333.228,E2 -12333.228} C_VEL
LIN {X 0,Y 374.554,Z 551.579,A -85,B 0,C 180,E1 -12334.304,E2 -12334.304} C_VEL
LIN {X 0,Y 374.568,Z 548.373,A -85,B 0,C 180,E1 -12336.045,E2 -12336.045} C_VEL
LIN {X 0,Y 374.808,Z 544.656,A -85,B 0,C 180,E1 -12337.542,E2 -12337.542} C_VEL
LIN {X 0,Y 375.248,Z 538.538,A -85,B 0,C 180,E1 -12339.432,E2 -12339.432} C_VEL
LIN {X 0,Y 375.813,Z 531.855,A -85,B 0,C 180,E1 -12341.051,E2 -12341.051} C_VEL
LIN {X 0,Y 376.714,Z 523.57,A -85,B 0,C 180,E1 -12342.662,E2 -12342.662} C_VEL
LIN {X 0,Y 377.542,Z 515.075,A -85,B 0,C 180,E1 -12344.004,E2 -12344.004} C_VEL
LIN {X 0,Y 378.515,Z 504.578,A -85,B 0,C 180,E1 -12345.342,E2 -12345.342} C_VEL
LIN {X 0,Y 379.601,Z 492.767,A -85,B 0,C 180,E1 -12346.538,E2 -12346.538} C_VEL
LIN {X 0,Y 380.432,Z 482.009,A -85,B 0,C 180,E1 -12347.391,E2 -12347.391} C_VEL
LIN {X 0,Y 379.123,Z 470.101,A -85,B 0,C 180,E1 -12348.211,E2 -12348.211} C_VEL
LIN {X 0,Y 377.186,Z 458.071,A -85,B 0,C 180,E1 -12348.867,E2 -12348.867} C_VEL
LIN {X 0,Y 375.202,Z 448.109,A -85,B 0,C 180,E1 -12349.312,E2 -12349.312} C_VEL
LIN {X 0,Y 375.559,Z 442.114,A -85,B 0,C 180,E1 -12352.558,E2 -12352.558} C_VEL
LIN {X 0,Y 375.98,Z 435.425,A -85,B 0,C 180,E1 -12356.202,E2 -12356.202} C_VEL
LIN {X 0,Y 376.564,Z 429.216,A -85,B 0,C 180,E1 -12359.642,E2 -12359.642} C_VEL
LIN {X 0,Y 377.039,Z 423.361,A -85,B 0,C 180,E1 -12362.986,E2 -12362.986} C_VEL
LIN {X 0,Y 377.355,Z 418.421,A -85,B 0,C 180,E1 -12365.921,E2 -12365.921} C_VEL
LIN {X 0,Y 377.001,Z 414.399,A -85,B 0,C 180,E1 -12368.468,E2 -12368.468} C_VEL
LIN {X 0,Y 376.164,Z 409.695,A -85,B 0,C 180,E1 -12371.64,E2 -12371.64} C_VEL
LIN {X 0,Y 375.968,Z 408.658,A -85,B 0,C 180,E1 -12372.468,E2 -12372.468} C_VEL
LIN {X 0,Y 375.931,Z 408.658,A -85,B 0,C 180,E1 -12376.234,E2 -12376.234} C_VEL
LIN {X 0,Y 375.99,Z 408.647,A -85,B 0,C 180,E1 -12380.029,E2 -12380.029} C_VEL
LIN {X 0,Y 375.966,Z 408.651,A -85,B 0,C 180,E1 -12383.495,E2 -12383.495} C_VEL
LIN {X 0,Y 375.961,Z 408.651,A -85,B 0,C 180,E1 -12385.889,E2 -12385.889} C_VEL
LIN {X 0,Y 375.966,Z 408.65,A -85,B 0,C 180,E1 -12389.687,E2 -12389.687} C_VEL
LIN {X 0,Y 376.021,Z 408.644,A -85,B 0,C 180,E1 -12393.348,E2 -12393.348} C_VEL
LIN {X 0,Y 375.997,Z 408.65,A -85,B 0,C 180,E1 -12396.888,E2 -12396.888} C_VEL
LIN {X 0,Y 375.999,Z 408.65,A -85,B 0,C 180,E1 -12400.339,E2 -12400.339} C_VEL
LIN {X 0,Y 376.031,Z 408.642,A -85,B 0,C 180,E1 -12403.719,E2 -12403.719} C_VEL
LIN {X 0,Y 376.108,Z 408.633,A -85,B 0,C 180,E1 -12407.042,E2 -12407.042} C_VEL
LIN {X 0,Y 376.126,Z 408.636,A -85,B 0,C 180,E1 -12410.319,E2 -12410.319} C_VEL
LIN {X 0,Y 376.232,Z 408.622,A -85,B 0,C 180,E1 -12412.487,E2 -12412.487} C_VEL
LIN {X 0,Y 376.173,Z 408.627,A -85,B 0,C 180,E1 -12414.64,E2 -12414.64} C_VEL
LIN {X 0,Y 376.353,Z 408.604,A -85,B 0,C 180,E1 -12417.86,E2 -12417.86} C_VEL
LIN {X 0,Y 376.491,Z 408.588,A -85,B 0,C 180,E1 -12420,E2 -12420} C_VEL
LIN {X 0,Y 376.186,Z 408.623,A -85,B 0,C 180,E1 -12423.213,E2 -12423.213} C_VEL
LIN {X 0,Y 376.235,Z 408.618,A -85,B 0,C 180,E1 -12426.636,E2 -12426.636} C_VEL
LIN {X 0,Y 376.208,Z 408.621,A -85,B 0,C 180,E1 -12428.595,E2 -12428.595} C_VEL
LIN {X 0,Y 376.061,Z 408.643,A -85,B 0,C 180,E1 -12431.863,E2 -12431.863} C_VEL
LIN {X 0,Y 376.062,Z 408.638,A -85,B 0,C 180,E1 -12435.167,E2 -12435.167} C_VEL
LIN {X 0,Y 376.01,Z 408.645,A -85,B 0,C 180,E1 -12438.527,E2 -12438.527} C_VEL
LIN {X 0,Y 375.964,Z 408.655,A -85,B 0,C 180,E1 -12441.954,E2 -12441.954} C_VEL
LIN {X 0,Y 376.008,Z 408.648,A -85,B 0,C 180,E1 -12445.461,E2 -12445.461} C_VEL
LIN {X 0,Y 375.963,Z 408.652,A -85,B 0,C 180,E1 -12449.08,E2 -12449.08} C_VEL
LIN {X 0,Y 375.952,Z 408.652,A -85,B 0,C 180,E1 -12452.828,E2 -12452.828} C_VEL
LIN {X 0,Y 375.96,Z 408.656,A -85,B 0,C 180,E1 -12455.415,E2 -12455.415} C_VEL
LIN {X 0,Y 375.978,Z 408.648,A -85,B 0,C 180,E1 -12458.271,E2 -12458.271} C_VEL
LIN {X 0,Y 375.937,Z 408.658,A -85,B 0,C 180,E1 -12461.601,E2 -12461.601} C_VEL
LIN {X 0,Y 375.956,Z 408.657,A -85,B 0,C 180,E1 -12465.265,E2 -12465.265} C_VEL
LIN {X 0,Y 375.942,Z 408.658,A -85,B 0,C 180,E1 -12469.133,E2 -12469.133} C_VEL
LIN {X 0,Y 375.961,Z 408.656,A -85,B 0,C 180,E1 -12471.911,E2 -12471.911} C_VEL
LIN {X 0,Y 375.89,Z 408.665,A -85,B 0,C 180,E1 -12473.511,E2 -12473.511} C_VEL
LIN {X 0,Y 375.898,Z 410.264,A -85,B 0,C 180,E1 -12475.351,E2 -12475.351} C_VEL
LIN {X 0,Y 375.727,Z 413.738,A -85,B 0,C 180,E1 -12478.416,E2 -12478.416} C_VEL
LIN {X 0,Y 375.483,Z 418.047,A -85,B 0,C 180,E1 -12482.1,E2 -12482.1} C_VEL
LIN {X 0,Y 375.333,Z 420.961,A -85,B 0,C 180,E1 -12484.49,E2 -12484.49} C_VEL
LIN {X 0,Y 375.091,Z 425.336,A -85,B 0,C 180,E1 -12487.992,E2 -12487.992} C_VEL
LIN {X 0,Y 375.013,Z 428.967,A -85,B 0,C 180,E1 -12490.775,E2 -12490.775} C_VEL
LIN {X 0,Y 378.274,Z 441.922,A -85,B 0,C 180,E1 -12491.416,E2 -12491.416} C_VEL
LIN {X 0,Y 380.754,Z 454.096,A -85,B 0,C 180,E1 -12492.195,E2 -12492.195} C_VEL
LIN {X 0,Y 381.191,Z 458.187,A -85,B 0,C 180,E1 -12492.485,E2 -12492.485} C_VEL
LIN {X 0,Y 380.319,Z 469.782,A -85,B 0,C 180,E1 -12493.356,E2 -12493.356} C_VEL
LIN {X 0,Y 379.496,Z 480.317,A -85,B 0,C 180,E1 -12494.367,E2 -12494.367} C_VEL
LIN {X 0,Y 378.681,Z 489.783,A -85,B 0,C 180,E1 -12495.49,E2 -12495.49} C_VEL
LIN {X 0,Y 377.675,Z 498.963,A -85,B 0,C 180,E1 -12496.823,E2 -12496.823} C_VEL
LIN {X 0,Y 376.768,Z 507.874,A -85,B 0,C 180,E1 -12498.432,E2 -12498.432} C_VEL
LIN {X 0,Y 376.015,Z 515.047,A -85,B 0,C 180,E1 -12500.044,E2 -12500.044} C_VEL
LIN {X 0,Y 375.449,Z 519.887,A -85,B 0,C 180,E1 -12501.388,E2 -12501.388} C_VEL
LIN {X 0,Y 375.046,Z 525.341,A -85,B 0,C 180,E1 -12503.302,E2 -12503.302} C_VEL
LIN {X 0,Y 374.881,Z 528.178,A -85,B 0,C 180,E1 -12504.621,E2 -12504.621} C_VEL
LIN {X 0,Y 374.685,Z 530.039,A -85,B 0,C 180,E1 -12505.697,E2 -12505.697} C_VEL
LIN {X 0,Y 374.587,Z 531.438,A -85,B 0,C 180,E1 -12506.773,E2 -12506.773} C_VEL
LIN {X 0,Y 374.569,Z 532.431,A -85,B 0,C 180,E1 -12507.85,E2 -12507.85} C_VEL
LIN {X 0,Y 374.555,Z 533.275,A -85,B 0,C 180,E1 -12510,E2 -12510} C_VEL
LIN {X 0,Y 374.546,Z 533.086,A -85,B 0,C 180,E1 -12511.075,E2 -12511.075} C_VEL
LIN {X 0,Y 374.568,Z 532.502,A -85,B 0,C 180,E1 -12512.151,E2 -12512.151} C_VEL
LIN {X 0,Y 374.677,Z 530.181,A -85,B 0,C 180,E1 -12514.303,E2 -12514.303} C_VEL
LIN {X 0,Y 374.946,Z 527.313,A -85,B 0,C 180,E1 -12515.917,E2 -12515.917} C_VEL
LIN {X 0,Y 375.181,Z 523.43,A -85,B 0,C 180,E1 -12517.535,E2 -12517.535} C_VEL
LIN {X 0,Y 375.638,Z 518.416,A -85,B 0,C 180,E1 -12519.151,E2 -12519.151} C_VEL
LIN {X 0,Y 376.287,Z 512.102,A -85,B 0,C 180,E1 -12520.765,E2 -12520.765} C_VEL
LIN {X 0,Y 377.096,Z 504.198,A -85,B 0,C 180,E1 -12522.376,E2 -12522.376} C_VEL
LIN {X 0,Y 378.172,Z 494.363,A -85,B 0,C 180,E1 -12523.981,E2 -12523.981} C_VEL
LIN {X 0,Y 379.154,Z 484.197,A -85,B 0,C 180,E1 -12525.297,E2 -12525.297} C_VEL
LIN {X 0,Y 379.972,Z 473.816,A -85,B 0,C 180,E1 -12526.384,E2 -12526.384} C_VEL
LIN {X 0,Y 380.965,Z 461.852,A -85,B 0,C 180,E1 -12527.367,E2 -12527.367} C_VEL
LIN {X 0,Y 381.048,Z 456.192,A -85,B 0,C 180,E1 -12527.761,E2 -12527.761} C_VEL
LIN {X 0,Y 378.715,Z 444.272,A -85,B 0,C 180,E1 -12528.553,E2 -12528.553} C_VEL
LIN {X 0,Y 375.493,Z 431.09,A -85,B 0,C 180,E1 -12529.236,E2 -12529.236} C_VEL
LIN {X 0,Y 374.998,Z 428.927,A -85,B 0,C 180,E1 -12529.359,E2 -12529.359} C_VEL
LIN {X 0,Y 375.211,Z 423.727,A -85,B 0,C 180,E1 -12533.391,E2 -12533.391} C_VEL
LIN {X 0,Y 375.209,Z 423.637,A -85,B 0,C 180,E1 -12533.464,E2 -12533.464} C_VEL
LIN {X 0,Y 374.542,Z 422.617,A -85,B 0,C 180,E1 -12534.347,E2 -12534.347} C_VEL
LIN {X 0,Y 371.748,Z 421.168,A -85,B 0,C 180,E1 -12535.792,E2 -12535.792} C_VEL
LIN {X 0,Y 369.43,Z 420.03,A -85,B 0,C 180,E1 -12536.96,E2 -12536.96} C_VEL
LIN {X 0,Y 368.489,Z 419.071,A -85,B 0,C 180,E1 -12537.86,E2 -12537.86} C_VEL
LIN {X 0,Y 368.441,Z 418.718,A -85,B 0,C 180,E1 -12538.164,E2 -12538.164} C_VEL
LIN {X 0,Y 368.641,Z 415.462,A -85,B 0,C 180,E1 -12540.981,E2 -12540.981} C_VEL
LIN {X 0,Y 368.769,Z 412.573,A -85,B 0,C 180,E1 -12543.551,E2 -12543.551} C_VEL
LIN {X 0,Y 368.827,Z 409.664,A -85,B 0,C 180,E1 -12546.207,E2 -12546.207} C_VEL
LIN {X 0,Y 368.903,Z 409.535,A -85,B 0,C 180,E1 -12548.953,E2 -12548.953} C_VEL
LIN {X 0,Y 368.884,Z 409.532,A -85,B 0,C 180,E1 -12552.009,E2 -12552.009} C_VEL
LIN {X 0,Y 368.888,Z 409.533,A -85,B 0,C 180,E1 -12555.177,E2 -12555.177} C_VEL
LIN {X 0,Y 368.885,Z 409.534,A -85,B 0,C 180,E1 -12558.178,E2 -12558.178} C_VEL
LIN {X 0,Y 368.912,Z 409.529,A -85,B 0,C 180,E1 -12561.359,E2 -12561.359} C_VEL
LIN {X 0,Y 368.939,Z 409.526,A -85,B 0,C 180,E1 -12565.147,E2 -12565.147} C_VEL
LIN {X 0,Y 368.932,Z 409.527,A -85,B 0,C 180,E1 -12569.046,E2 -12569.046} C_VEL
LIN {X 0,Y 368.966,Z 409.524,A -85,B 0,C 180,E1 -12572.797,E2 -12572.797} C_VEL
LIN {X 0,Y 368.948,Z 409.528,A -85,B 0,C 180,E1 -12576.113,E2 -12576.113} C_VEL
LIN {X 0,Y 368.939,Z 409.528,A -85,B 0,C 180,E1 -12579.947,E2 -12579.947} C_VEL
LIN {X 0,Y 368.979,Z 409.521,A -85,B 0,C 180,E1 -12583.399,E2 -12583.399} C_VEL
LIN {X 0,Y 369.061,Z 409.51,A -85,B 0,C 180,E1 -12586.79,E2 -12586.79} C_VEL
LIN {X 0,Y 369.071,Z 409.514,A -85,B 0,C 180,E1 -12590.132,E2 -12590.132} C_VEL
LIN {X 0,Y 369.191,Z 409.496,A -85,B 0,C 180,E1 -12592.342,E2 -12592.342} C_VEL
LIN {X 0,Y 369.147,Z 409.5,A -85,B 0,C 180,E1 -12594.538,E2 -12594.538} C_VEL
LIN {X 0,Y 369.319,Z 409.484,A -85,B 0,C 180,E1 -12597.819,E2 -12597.819} C_VEL
LIN {X 0,Y 369.46,Z 409.465,A -85,B 0,C 180,E1 -12600,E2 -12600} C_VEL
LIN {X 0,Y 369.32,Z 409.48,A -85,B 0,C 180,E1 -12602.181,E2 -12602.181} C_VEL
LIN {X 0,Y 369.212,Z 409.491,A -85,B 0,C 180,E1 -12606.558,E2 -12606.558} C_VEL
LIN {X 0,Y 369.142,Z 409.5,A -85,B 0,C 180,E1 -12608.761,E2 -12608.761} C_VEL
LIN {X 0,Y 369.016,Z 409.517,A -85,B 0,C 180,E1 -12612.093,E2 -12612.093} C_VEL
LIN {X 0,Y 369.002,Z 409.523,A -85,B 0,C 180,E1 -12615.465,E2 -12615.465} C_VEL
LIN {X 0,Y 368.961,Z 409.524,A -85,B 0,C 180,E1 -12618.894,E2 -12618.894} C_VEL
LIN {X 0,Y 368.935,Z 409.526,A -85,B 0,C 180,E1 -12622.395,E2 -12622.395} C_VEL
LIN {X 0,Y 369.002,Z 409.518,A -85,B 0,C 180,E1 -12625.98,E2 -12625.98} C_VEL
LIN {X 0,Y 368.917,Z 409.53,A -85,B 0,C 180,E1 -12629.69,E2 -12629.69} C_VEL
LIN {X 0,Y 368.899,Z 409.535,A -85,B 0,C 180,E1 -12633.043,E2 -12633.043} C_VEL
LIN {X 0,Y 368.92,Z 409.527,A -85,B 0,C 180,E1 -12636.197,E2 -12636.197} C_VEL
LIN {X 0,Y 368.907,Z 409.535,A -85,B 0,C 180,E1 -12638.953,E2 -12638.953} C_VEL
LIN {X 0,Y 368.883,Z 409.532,A -85,B 0,C 180,E1 -12642.009,E2 -12642.009} C_VEL
LIN {X 0,Y 368.888,Z 409.536,A -85,B 0,C 180,E1 -12645.177,E2 -12645.177} C_VEL
LIN {X 0,Y 368.964,Z 409.643,A -85,B 0,C 180,E1 -12647.38,E2 -12647.38} C_VEL
LIN {X 0,Y 369.721,Z 414.031,A -85,B 0,C 180,E1 -12650.446,E2 -12650.446} C_VEL
LIN {X 0,Y 370.227,Z 417.682,A -85,B 0,C 180,E1 -12652.872,E2 -12652.872} C_VEL
LIN {X 0,Y 370.393,Z 420.538,A -85,B 0,C 180,E1 -12654.677,E2 -12654.677} C_VEL
LIN {X 0,Y 369.848,Z 425.862,A -85,B 0,C 180,E1 -12657.855,E2 -12657.855} C_VEL
LIN {X 0,Y 369.375,Z 431.42,A -85,B 0,C 180,E1 -12661.072,E2 -12661.072} C_VEL
LIN {X 0,Y 368.757,Z 438.744,A -85,B 0,C 180,E1 -12665.21,E2 -12665.21} C_VEL
LIN {X 0,Y 368.325,Z 445.103,A -85,B 0,C 180,E1 -12668.744,E2 -12668.744} C_VEL
LIN {X 0,Y 368.178,Z 448.112,A -85,B 0,C 180,E1 -12670.322,E2 -12670.322} C_VEL
LIN {X 0,Y 370.858,Z 461.309,A -85,B 0,C 180,E1 -12670.926,E2 -12670.926} C_VEL
LIN {X 0,Y 372.729,Z 474.057,A -85,B 0,C 180,E1 -12671.701,E2 -12671.701} C_VEL
LIN {X 0,Y 373.595,Z 483.287,A -85,B 0,C 180,E1 -12672.385,E2 -12672.385} C_VEL
LIN {X 0,Y 372.567,Z 495.52,A -85,B 0,C 180,E1 -12673.422,E2 -12673.422} C_VEL
LIN {X 0,Y 371.552,Z 505.633,A -85,B 0,C 180,E1 -12674.503,E2 -12674.503} C_VEL
LIN {X 0,Y 370.633,Z 514.934,A -85,B 0,C 180,E1 -12675.729,E2 -12675.729} C_VEL
LIN {X 0,Y 369.772,Z 523.415,A -85,B 0,C 180,E1 -12677.096,E2 -12677.096} C_VEL
LIN {X 0,Y 368.819,Z 531.69,A -85,B 0,C 180,E1 -12678.737,E2 -12678.737} C_VEL
LIN {X 0,Y 368.221,Z 538.366,A -85,B 0,C 180,E1 -12680.386,E2 -12680.386} C_VEL
LIN {X 0,Y 367.734,Z 544.475,A -85,B 0,C 180,E1 -12682.312,E2 -12682.312} C_VEL
LIN {X 0,Y 367.469,Z 548.523,A -85,B 0,C 180,E1 -12684.001,E2 -12684.001} C_VEL
LIN {X 0,Y 367.459,Z 551.383,A -85,B 0,C 180,E1 -12685.612,E2 -12685.612} C_VEL
LIN {X 0,Y 367.381,Z 552.779,A -85,B 0,C 180,E1 -12686.71,E2 -12686.71} C_VEL
LIN {X 0,Y 367.417,Z 554.385,A -85,B 0,C 180,E1 -12688.904,E2 -12688.904} C_VEL
LIN {X 0,Y 367.456,Z 554.602,A -85,B 0,C 180,E1 -12690,E2 -12690} C_VEL
LIN {X 0,Y 367.417,Z 554.382,A -85,B 0,C 180,E1 -12691.096,E2 -12691.096} C_VEL
LIN {X 0,Y 367.381,Z 552.773,A -85,B 0,C 180,E1 -12693.29,E2 -12693.29} C_VEL
LIN {X 0,Y 367.459,Z 551.374,A -85,B 0,C 180,E1 -12694.388,E2 -12694.388} C_VEL
LIN {X 0,Y 367.477,Z 548.483,A -85,B 0,C 180,E1 -12696.01,E2 -12696.01} C_VEL
LIN {X 0,Y 367.734,Z 544.45,A -85,B 0,C 180,E1 -12697.688,E2 -12697.688} C_VEL
LIN {X 0,Y 368.22,Z 538.332,A -85,B 0,C 180,E1 -12699.614,E2 -12699.614} C_VEL
LIN {X 0,Y 368.818,Z 531.648,A -85,B 0,C 180,E1 -12701.263,E2 -12701.263} C_VEL
LIN {X 0,Y 369.772,Z 523.363,A -85,B 0,C 180,E1 -12702.904,E2 -12702.904} C_VEL
LIN {X 0,Y 370.787,Z 513.66,A -85,B 0,C 180,E1 -12704.439,E2 -12704.439} C_VEL
LIN {X 0,Y 371.72,Z 503.192,A -85,B 0,C 180,E1 -12705.77,E2 -12705.77} C_VEL
LIN {X 0,Y 372.792,Z 492.559,A -85,B 0,C 180,E1 -12706.849,E2 -12706.849} C_VEL
LIN {X 0,Y 373.54,Z 481.938,A -85,B 0,C 180,E1 -12707.712,E2 -12707.712} C_VEL
LIN {X 0,Y 372.273,Z 470.651,A -85,B 0,C 180,E1 -12708.516,E2 -12708.516} C_VEL
LIN {X 0,Y 370.234,Z 458.204,A -85,B 0,C 180,E1 -12709.221,E2 -12709.221} C_VEL
LIN {X 0,Y 368.165,Z 447.911,A -85,B 0,C 180,E1 -12709.696,E2 -12709.696} C_VEL
LIN {X 0,Y 368.542,Z 441.924,A -85,B 0,C 180,E1 -12713.012,E2 -12713.012} C_VEL
LIN {X 0,Y 368.949,Z 435.747,A -85,B 0,C 180,E1 -12716.454,E2 -12716.454} C_VEL
LIN {X 0,Y 369.53,Z 430.139,A -85,B 0,C 180,E1 -12719.636,E2 -12719.636} C_VEL
LIN {X 0,Y 370.064,Z 423.646,A -85,B 0,C 180,E1 -12723.418,E2 -12723.418} C_VEL
LIN {X 0,Y 370.341,Z 419.344,A -85,B 0,C 180,E1 -12726.036,E2 -12726.036} C_VEL
LIN {X 0,Y 369.915,Z 415.043,A -85,B 0,C 180,E1 -12728.835,E2 -12728.835} C_VEL
LIN {X 0,Y 369.088,Z 410.418,A -85,B 0,C 180,E1 -12732.045,E2 -12732.045} C_VEL
LIN {X 0,Y 368.943,Z 409.531,A -85,B 0,C 180,E1 -12732.79,E2 -12732.79} C_VEL
LIN {X 0,Y 368.887,Z 409.536,A -85,B 0,C 180,E1 -12736.696,E2 -12736.696} C_VEL
LIN {X 0,Y 368.913,Z 409.529,A -85,B 0,C 180,E1 -12739.643,E2 -12739.643} C_VEL
LIN {X 0,Y 368.904,Z 409.534,A -85,B 0,C 180,E1 -12743.144,E2 -12743.144} C_VEL
LIN {X 0,Y 368.897,Z 409.533,A -85,B 0,C 180,E1 -12746.462,E2 -12746.462} C_VEL
LIN {X 0,Y 368.93,Z 409.53,A -85,B 0,C 180,E1 -12749.046,E2 -12749.046} C_VEL
LIN {X 0,Y 368.964,Z 409.528,A -85,B 0,C 180,E1 -12752.797,E2 -12752.797} C_VEL
LIN {X 0,Y 368.946,Z 409.525,A -85,B 0,C 180,E1 -12756.113,E2 -12756.113} C_VEL
LIN {X 0,Y 368.938,Z 409.526,A -85,B 0,C 180,E1 -12759.947,E2 -12759.947} C_VEL
LIN {X 0,Y 368.977,Z 409.52,A -85,B 0,C 180,E1 -12763.399,E2 -12763.399} C_VEL
LIN {X 0,Y 369.061,Z 409.513,A -85,B 0,C 180,E1 -12766.79,E2 -12766.79} C_VEL
LIN {X 0,Y 369.074,Z 409.512,A -85,B 0,C 180,E1 -12770.132,E2 -12770.132} C_VEL
LIN {X 0,Y 369.19,Z 409.5,A -85,B 0,C 180,E1 -12772.342,E2 -12772.342} C_VEL
LIN {X 0,Y 369.146,Z 409.504,A -85,B 0,C 180,E1 -12774.538,E2 -12774.538} C_VEL
LIN {X 0,Y 369.318,Z 409.48,A -85,B 0,C 180,E1 -12777.819,E2 -12777.819} C_VEL
LIN {X 0,Y 369.46,Z 409.464,A -85,B 0,C 180,E1 -12780,E2 -12780} C_VEL
LIN {X 0,Y 369.318,Z 409.484,A -85,B 0,C 180,E1 -12782.181,E2 -12782.181} C_VEL
LIN {X 0,Y 369.205,Z 409.493,A -85,B 0,C 180,E1 -12786.624,E2 -12786.624} C_VEL
LIN {X 0,Y 369.141,Z 409.5,A -85,B 0,C 180,E1 -12788.761,E2 -12788.761} C_VEL
LIN {X 0,Y 369.015,Z 409.521,A -85,B 0,C 180,E1 -12792.093,E2 -12792.093} C_VEL
LIN {X 0,Y 369,Z 409.519,A -85,B 0,C 180,E1 -12795.465,E2 -12795.465} C_VEL
LIN {X 0,Y 368.959,Z 409.523,A -85,B 0,C 180,E1 -12798.894,E2 -12798.894} C_VEL
LIN {X 0,Y 368.934,Z 409.527,A -85,B 0,C 180,E1 -12802.395,E2 -12802.395} C_VEL
LIN {X 0,Y 369.001,Z 409.521,A -85,B 0,C 180,E1 -12805.98,E2 -12805.98} C_VEL
LIN {X 0,Y 368.916,Z 409.534,A -85,B 0,C 180,E1 -12809.69,E2 -12809.69} C_VEL
LIN {X 0,Y 368.9,Z 409.531,A -85,B 0,C 180,E1 -12813.044,E2 -12813.044} C_VEL
LIN {X 0,Y 368.92,Z 409.528,A -85,B 0,C 180,E1 -12816.197,E2 -12816.197} C_VEL
LIN {X 0,Y 368.907,Z 409.531,A -85,B 0,C 180,E1 -12818.953,E2 -12818.953} C_VEL
LIN {X 0,Y 368.883,Z 409.533,A -85,B 0,C 180,E1 -12822.01,E2 -12822.01} C_VEL
LIN {X 0,Y 368.929,Z 409.531,A -85,B 0,C 180,E1 -12825.183,E2 -12825.183} C_VEL
LIN {X 0,Y 368.885,Z 409.532,A -85,B 0,C 180,E1 -12828.178,E2 -12828.178} C_VEL
LIN {X 0,Y 368.907,Z 409.535,A -85,B 0,C 180,E1 -12831.36,E2 -12831.36} C_VEL
LIN {X 0,Y 368.803,Z 409.548,A -85,B 0,C 180,E1 -12833.79,E2 -12833.79} C_VEL
LIN {X 0,Y 368.767,Z 412.446,A -85,B 0,C 180,E1 -12836.449,E2 -12836.449} C_VEL
LIN {X 0,Y 368.644,Z 415.415,A -85,B 0,C 180,E1 -12839.082,E2 -12839.082} C_VEL
LIN {X 0,Y 368.381,Z 419.677,A -85,B 0,C 180,E1 -12842.75,E2 -12842.75} C_VEL
LIN {X 0,Y 368.159,Z 424.091,A -85,B 0,C 180,E1 -12846.392,E2 -12846.392} C_VEL
LIN {X 0,Y 367.964,Z 429.188,A -85,B 0,C 180,E1 -12850.392,E2 -12850.392} C_VEL
LIN {X 0,Y 371.217,Z 442.001,A -85,B 0,C 180,E1 -12851.043,E2 -12851.043} C_VEL
LIN {X 0,Y 373.85,Z 454.837,A -85,B 0,C 180,E1 -12851.888,E2 -12851.888} C_VEL
LIN {X 0,Y 374.337,Z 459.881,A -85,B 0,C 180,E1 -12852.259,E2 -12852.259} C_VEL
LIN {X 0,Y 373.38,Z 471.562,A -85,B 0,C 180,E1 -12853.178,E2 -12853.178} C_VEL
LIN {X 0,Y 372.532,Z 482.386,A -85,B 0,C 180,E1 -12854.283,E2 -12854.283} C_VEL
LIN {X 0,Y 371.599,Z 491.948,A -85,B 0,C 180,E1 -12855.487,E2 -12855.487} C_VEL
LIN {X 0,Y 370.557,Z 500.791,A -85,B 0,C 180,E1 -12856.845,E2 -12856.845} C_VEL
LIN {X 0,Y 369.641,Z 509.412,A -85,B 0,C 180,E1 -12858.484,E2 -12858.484} C_VEL
LIN {X 0,Y 368.886,Z 516.284,A -85,B 0,C 180,E1 -12860.127,E2 -12860.127} C_VEL
LIN {X 0,Y 368.273,Z 521.786,A -85,B 0,C 180,E1 -12861.771,E2 -12861.771} C_VEL
LIN {X 0,Y 367.97,Z 526.101,A -85,B 0,C 180,E1 -12863.42,E2 -12863.42} C_VEL
LIN {X 0,Y 367.812,Z 528.383,A -85,B 0,C 180,E1 -12864.518,E2 -12864.518} C_VEL
LIN {X 0,Y 367.62,Z 530.243,A -85,B 0,C 180,E1 -12865.614,E2 -12865.614} C_VEL
LIN {X 0,Y 367.501,Z 531.642,A -85,B 0,C 180,E1 -12866.711,E2 -12866.711} C_VEL
LIN {X 0,Y 367.45,Z 533.247,A -85,B 0,C 180,E1 -12868.904,E2 -12868.904} C_VEL
LIN {X 0,Y 367.458,Z 533.479,A -85,B 0,C 180,E1 -12870,E2 -12870} C_VEL
LIN {X 0,Y 367.45,Z 533.29,A -85,B 0,C 180,E1 -12871.096,E2 -12871.096} C_VEL
LIN {X 0,Y 367.471,Z 532.706,A -85,B 0,C 180,E1 -12872.192,E2 -12872.192} C_VEL
LIN {X 0,Y 367.613,Z 530.384,A -85,B 0,C 180,E1 -12874.386,E2 -12874.386} C_VEL
LIN {X 0,Y 367.884,Z 527.068,A -85,B 0,C 180,E1 -12876.249,E2 -12876.249} C_VEL
LIN {X 0,Y 368.271,Z 522.076,A -85,B 0,C 180,E1 -12878.229,E2 -12878.229} C_VEL
LIN {X 0,Y 368.998,Z 515.639,A -85,B 0,C 180,E1 -12880.147,E2 -12880.147} C_VEL
LIN {X 0,Y 369.713,Z 508.567,A -85,B 0,C 180,E1 -12881.792,E2 -12881.792} C_VEL
LIN {X 0,Y 370.698,Z 499.752,A -85,B 0,C 180,E1 -12883.429,E2 -12883.429} C_VEL
LIN {X 0,Y 371.747,Z 490.702,A -85,B 0,C 180,E1 -12884.787,E2 -12884.787} C_VEL
LIN {X 0,Y 372.585,Z 480.641,A -85,B 0,C 180,E1 -12886.019,E2 -12886.019} C_VEL
LIN {X 0,Y 373.598,Z 469.537,A -85,B 0,C 180,E1 -12887.094,E2 -12887.094} C_VEL
LIN {X 0,Y 374.342,Z 458.147,A -85,B 0,C 180,E1 -12887.966,E2 -12887.966} C_VEL
LIN {X 0,Y 372.425,Z 447.689,A -85,B 0,C 180,E1 -12888.712,E2 -12888.712} C_VEL
LIN {X 0,Y 369.409,Z 434.854,A -85,B 0,C 180,E1 -12889.451,E2 -12889.451} C_VEL
LIN {X 0,Y 367.953,Z 429.177,A -85,B 0,C 180,E1 -12889.712,E2 -12889.712} C_VEL
LIN {X 0,Y 368.172,Z 424.196,A -85,B 0,C 180,E1 -12893.633,E2 -12893.633} C_VEL
LIN {X 0,Y 368.388,Z 419.811,A -85,B 0,C 180,E1 -12897.25,E2 -12897.25} C_VEL
LIN {X 0,Y 368.441,Z 418.718,A -85,B 0,C 180,E1 -12898.164,E2 -12898.164} C_VEL
LIN {X 0,Y 367.869,Z 417.74,A -85,B 0,C 180,E1 -12899.064,E2 -12899.064} C_VEL
LIN {X 0,Y 365.134,Z 416.411,A -85,B 0,C 180,E1 -12900.539,E2 -12900.539} C_VEL
LIN {X 0,Y 362.787,Z 415.384,A -85,B 0,C 180,E1 -12901.733,E2 -12901.733} C_VEL
LIN {X 0,Y 361.793,Z 414.487,A -85,B 0,C 180,E1 -12902.653,E2 -12902.653} C_VEL
LIN {X 0,Y 361.722,Z 414.153,A -85,B 0,C 180,E1 -12902.963,E2 -12902.963} C_VEL
LIN {X 0,Y 361.806,Z 411.263,A -85,B 0,C 180,E1 -12905.644,E2 -12905.644} C_VEL
LIN {X 0,Y 361.831,Z 410.414,A -85,B 0,C 180,E1 -12907.216,E2 -12907.216} C_VEL
LIN {X 0,Y 361.857,Z 410.407,A -85,B 0,C 180,E1 -12909.861,E2 -12909.861} C_VEL
LIN {X 0,Y 361.839,Z 410.415,A -85,B 0,C 180,E1 -12912.829,E2 -12912.829} C_VEL
LIN {X 0,Y 361.823,Z 410.412,A -85,B 0,C 180,E1 -12915.946,E2 -12915.946} C_VEL
LIN {X 0,Y 361.838,Z 410.41,A -85,B 0,C 180,E1 -12919.244,E2 -12919.244} C_VEL
LIN {X 0,Y 361.874,Z 410.409,A -85,B 0,C 180,E1 -12922.775,E2 -12922.775} C_VEL
LIN {X 0,Y 361.857,Z 410.407,A -85,B 0,C 180,E1 -12925.72,E2 -12925.72} C_VEL
LIN {X 0,Y 361.875,Z 410.405,A -85,B 0,C 180,E1 -12929.672,E2 -12929.672} C_VEL
LIN {X 0,Y 361.956,Z 410.395,A -85,B 0,C 180,E1 -12933.475,E2 -12933.475} C_VEL
LIN {X 0,Y 361.893,Z 410.403,A -85,B 0,C 180,E1 -12937.145,E2 -12937.145} C_VEL
LIN {X 0,Y 361.909,Z 410.402,A -85,B 0,C 180,E1 -12940.723,E2 -12940.723} C_VEL
LIN {X 0,Y 361.936,Z 410.397,A -85,B 0,C 180,E1 -12943.066,E2 -12943.066} C_VEL
LIN {X 0,Y 362.002,Z 410.391,A -85,B 0,C 180,E1 -12946.528,E2 -12946.528} C_VEL
LIN {X 0,Y 362.034,Z 410.39,A -85,B 0,C 180,E1 -12949.938,E2 -12949.938} C_VEL
LIN {X 0,Y 362.154,Z 410.374,A -85,B 0,C 180,E1 -12952.193,E2 -12952.193} C_VEL
LIN {X 0,Y 362.121,Z 410.376,A -85,B 0,C 180,E1 -12954.431,E2 -12954.431} C_VEL
LIN {X 0,Y 362.283,Z 410.359,A -85,B 0,C 180,E1 -12957.776,E2 -12957.776} C_VEL
LIN {X 0,Y 362.429,Z 410.34,A -85,B 0,C 180,E1 -12960,E2 -12960} C_VEL
LIN {X 0,Y 362.284,Z 410.356,A -85,B 0,C 180,E1 -12962.223,E2 -12962.223} C_VEL
LIN {X 0,Y 362.175,Z 410.367,A -85,B 0,C 180,E1 -12966.686,E2 -12966.686} C_VEL
LIN {X 0,Y 362.078,Z 410.38,A -85,B 0,C 180,E1 -12968.933,E2 -12968.933} C_VEL
LIN {X 0,Y 361.969,Z 410.393,A -85,B 0,C 180,E1 -12972.332,E2 -12972.332} C_VEL
LIN {X 0,Y 361.965,Z 410.394,A -85,B 0,C 180,E1 -12974.62,E2 -12974.62} C_VEL
LIN {X 0,Y 361.958,Z 410.395,A -85,B 0,C 180,E1 -12978.099,E2 -12978.099} C_VEL
LIN {X 0,Y 361.894,Z 410.406,A -85,B 0,C 180,E1 -12981.653,E2 -12981.653} C_VEL
LIN {X 0,Y 361.931,Z 410.404,A -85,B 0,C 180,E1 -12985.29,E2 -12985.29} C_VEL
LIN {X 0,Y 361.911,Z 410.402,A -85,B 0,C 180,E1 -12987.779,E2 -12987.779} C_VEL
LIN {X 0,Y 361.84,Z 410.411,A -85,B 0,C 180,E1 -12991.629,E2 -12991.629} C_VEL
LIN {X 0,Y 361.877,Z 410.408,A -85,B 0,C 180,E1 -12995.345,E2 -12995.345} C_VEL
LIN {X 0,Y 361.873,Z 410.411,A -85,B 0,C 180,E1 -12999.027,E2 -12999.027} C_VEL
LIN {X 0,Y 361.838,Z 410.414,A -85,B 0,C 180,E1 -13002.829,E2 -13002.829} C_VEL
LIN {X 0,Y 361.857,Z 410.413,A -85,B 0,C 180,E1 -13006.411,E2 -13006.411} C_VEL
LIN {X 0,Y 361.873,Z 410.428,A -85,B 0,C 180,E1 -13006.986,E2 -13006.986} C_VEL
LIN {X 0,Y 362.663,Z 414.967,A -85,B 0,C 180,E1 -13010.245,E2 -13010.245} C_VEL
LIN {X 0,Y 363.243,Z 419.26,A -85,B 0,C 180,E1 -13013.145,E2 -13013.145} C_VEL
LIN {X 0,Y 363.294,Z 422.487,A -85,B 0,C 180,E1 -13015.202,E2 -13015.202} C_VEL
LIN {X 0,Y 362.633,Z 428.955,A -85,B 0,C 180,E1 -13019.11,E2 -13019.11} C_VEL
LIN {X 0,Y 362.098,Z 434.298,A -85,B 0,C 180,E1 -13022.237,E2 -13022.237} C_VEL
LIN {X 0,Y 361.569,Z 440.857,A -85,B 0,C 180,E1 -13026.003,E2 -13026.003} C_VEL
LIN {X 0,Y 361.165,Z 447.005,A -85,B 0,C 180,E1 -13029.496,E2 -13029.496} C_VEL
LIN {X 0,Y 361.117,Z 447.723,A -85,B 0,C 180,E1 -13029.903,E2 -13029.903} C_VEL
LIN {X 0,Y 364.063,Z 462.226,A -85,B 0,C 180,E1 -13030.61,E2 -13030.61} C_VEL
LIN {X 0,Y 365.967,Z 475.334,A -85,B 0,C 180,E1 -13031.446,E2 -13031.446} C_VEL
LIN {X 0,Y 366.735,Z 484.307,A -85,B 0,C 180,E1 -13032.144,E2 -13032.144} C_VEL
LIN {X 0,Y 365.609,Z 496.741,A -85,B 0,C 180,E1 -13033.241,E2 -13033.241} C_VEL
LIN {X 0,Y 364.564,Z 506.564,A -85,B 0,C 180,E1 -13034.342,E2 -13034.342} C_VEL
LIN {X 0,Y 363.523,Z 516.529,A -85,B 0,C 180,E1 -13035.73,E2 -13035.73} C_VEL
LIN {X 0,Y 362.636,Z 524.703,A -85,B 0,C 180,E1 -13037.122,E2 -13037.122} C_VEL
LIN {X 0,Y 361.681,Z 532.724,A -85,B 0,C 180,E1 -13038.795,E2 -13038.795} C_VEL
LIN {X 0,Y 361.087,Z 539.159,A -85,B 0,C 180,E1 -13040.477,E2 -13040.477} C_VEL
LIN {X 0,Y 360.684,Z 544.272,A -85,B 0,C 180,E1 -13042.16,E2 -13042.16} C_VEL
LIN {X 0,Y 360.379,Z 548.615,A -85,B 0,C 180,E1 -13044.038,E2 -13044.038} C_VEL
LIN {X 0,Y 360.367,Z 551.179,A -85,B 0,C 180,E1 -13045.526,E2 -13045.526} C_VEL
LIN {X 0,Y 360.301,Z 552.575,A -85,B 0,C 180,E1 -13046.645,E2 -13046.645} C_VEL
LIN {X 0,Y 360.317,Z 554.182,A -85,B 0,C 180,E1 -13048.882,E2 -13048.882} C_VEL
LIN {X 0,Y 360.359,Z 554.398,A -85,B 0,C 180,E1 -13050,E2 -13050} C_VEL
LIN {X 0,Y 360.317,Z 554.178,A -85,B 0,C 180,E1 -13051.118,E2 -13051.118} C_VEL
LIN {X 0,Y 360.301,Z 552.569,A -85,B 0,C 180,E1 -13053.355,E2 -13053.355} C_VEL
LIN {X 0,Y 360.367,Z 551.169,A -85,B 0,C 180,E1 -13054.474,E2 -13054.474} C_VEL
LIN {X 0,Y 360.378,Z 548.6,A -85,B 0,C 180,E1 -13055.961,E2 -13055.961} C_VEL
LIN {X 0,Y 360.684,Z 544.244,A -85,B 0,C 180,E1 -13057.839,E2 -13057.839} C_VEL
LIN {X 0,Y 361.194,Z 538.125,A -85,B 0,C 180,E1 -13059.803,E2 -13059.803} C_VEL
LIN {X 0,Y 361.835,Z 531.442,A -85,B 0,C 180,E1 -13061.484,E2 -13061.484} C_VEL
LIN {X 0,Y 362.835,Z 523.156,A -85,B 0,C 180,E1 -13063.155,E2 -13063.155} C_VEL
LIN {X 0,Y 363.758,Z 514.661,A -85,B 0,C 180,E1 -13064.547,E2 -13064.547} C_VEL
LIN {X 0,Y 364.767,Z 504.162,A -85,B 0,C 180,E1 -13065.935,E2 -13065.935} C_VEL
LIN {X 0,Y 365.98,Z 492.35,A -85,B 0,C 180,E1 -13067.172,E2 -13067.172} C_VEL
LIN {X 0,Y 366.706,Z 483.024,A -85,B 0,C 180,E1 -13067.95,E2 -13067.95} C_VEL
LIN {X 0,Y 365.394,Z 470.846,A -85,B 0,C 180,E1 -13068.855,E2 -13068.855} C_VEL
LIN {X 0,Y 363.316,Z 458.387,A -85,B 0,C 180,E1 -13069.586,E2 -13069.586} C_VEL
LIN {X 0,Y 361.117,Z 447.702,A -85,B 0,C 180,E1 -13070.097,E2 -13070.097} C_VEL
LIN {X 0,Y 361.445,Z 442.796,A -85,B 0,C 180,E1 -13072.885,E2 -13072.885} C_VEL
LIN {X 0,Y 361.937,Z 436.061,A -85,B 0,C 180,E1 -13076.719,E2 -13076.719} C_VEL
LIN {X 0,Y 362.555,Z 429.976,A -85,B 0,C 180,E1 -13080.265,E2 -13080.265} C_VEL
LIN {X 0,Y 363.163,Z 423.498,A -85,B 0,C 180,E1 -13084.14,E2 -13084.14} C_VEL
LIN {X 0,Y 363.319,Z 421.06,A -85,B 0,C 180,E1 -13085.665,E2 -13085.665} C_VEL
LIN {X 0,Y 363.036,Z 417.067,A -85,B 0,C 180,E1 -13088.279,E2 -13088.279} C_VEL
LIN {X 0,Y 362.304,Z 412.79,A -85,B 0,C 180,E1 -13091.264,E2 -13091.264} C_VEL
LIN {X 0,Y 361.875,Z 410.411,A -85,B 0,C 180,E1 -13093.013,E2 -13093.013} C_VEL
LIN {X 0,Y 361.837,Z 410.415,A -85,B 0,C 180,E1 -13097.171,E2 -13097.171} C_VEL
LIN {X 0,Y 361.872,Z 410.412,A -85,B 0,C 180,E1 -13100.973,E2 -13100.973} C_VEL
LIN {X 0,Y 361.876,Z 410.408,A -85,B 0,C 180,E1 -13104.655,E2 -13104.655} C_VEL
LIN {X 0,Y 361.838,Z 410.411,A -85,B 0,C 180,E1 -13108.371,E2 -13108.371} C_VEL
LIN {X 0,Y 361.909,Z 410.402,A -85,B 0,C 180,E1 -13112.221,E2 -13112.221} C_VEL
LIN {X 0,Y 361.929,Z 410.405,A -85,B 0,C 180,E1 -13114.71,E2 -13114.71} C_VEL
LIN {X 0,Y 361.893,Z 410.406,A -85,B 0,C 180,E1 -13118.347,E2 -13118.347} C_VEL
LIN {X 0,Y 361.968,Z 410.395,A -85,B 0,C 180,E1 -13122.061,E2 -13122.061} C_VEL
LIN {X 0,Y 362,Z 410.392,A -85,B 0,C 180,E1 -13126.101,E2 -13126.101} C_VEL
LIN {X 0,Y 362.038,Z 410.386,A -85,B 0,C 180,E1 -13129.938,E2 -13129.938} C_VEL
LIN {X 0,Y 362.153,Z 410.375,A -85,B 0,C 180,E1 -13132.193,E2 -13132.193} C_VEL
LIN {X 0,Y 362.119,Z 410.38,A -85,B 0,C 180,E1 -13134.431,E2 -13134.431} C_VEL
LIN {X 0,Y 362.282,Z 410.356,A -85,B 0,C 180,E1 -13137.776,E2 -13137.776} C_VEL
LIN {X 0,Y 362.43,Z 410.34,A -85,B 0,C 180,E1 -13140,E2 -13140} C_VEL
LIN {X 0,Y 362.282,Z 410.36,A -85,B 0,C 180,E1 -13142.224,E2 -13142.224} C_VEL
LIN {X 0,Y 362.174,Z 410.369,A -85,B 0,C 180,E1 -13146.686,E2 -13146.686} C_VEL
LIN {X 0,Y 362.077,Z 410.38,A -85,B 0,C 180,E1 -13148.933,E2 -13148.933} C_VEL
LIN {X 0,Y 361.969,Z 410.396,A -85,B 0,C 180,E1 -13152.332,E2 -13152.332} C_VEL
LIN {X 0,Y 361.964,Z 410.394,A -85,B 0,C 180,E1 -13154.62,E2 -13154.62} C_VEL
LIN {X 0,Y 361.957,Z 410.398,A -85,B 0,C 180,E1 -13158.1,E2 -13158.1} C_VEL
LIN {X 0,Y 361.893,Z 410.407,A -85,B 0,C 180,E1 -13161.653,E2 -13161.653} C_VEL
LIN {X 0,Y 361.93,Z 410.4,A -85,B 0,C 180,E1 -13165.29,E2 -13165.29} C_VEL
LIN {X 0,Y 361.91,Z 410.406,A -85,B 0,C 180,E1 -13167.779,E2 -13167.779} C_VEL
LIN {X 0,Y 361.839,Z 410.416,A -85,B 0,C 180,E1 -13171.629,E2 -13171.629} C_VEL
LIN {X 0,Y 361.876,Z 410.409,A -85,B 0,C 180,E1 -13175.345,E2 -13175.345} C_VEL
LIN {X 0,Y 361.873,Z 410.407,A -85,B 0,C 180,E1 -13179.027,E2 -13179.027} C_VEL
LIN {X 0,Y 361.838,Z 410.411,A -85,B 0,C 180,E1 -13182.829,E2 -13182.829} C_VEL
LIN {X 0,Y 361.837,Z 410.41,A -85,B 0,C 180,E1 -13185.944,E2 -13185.944} C_VEL
LIN {X 0,Y 361.838,Z 410.416,A -85,B 0,C 180,E1 -13189.245,E2 -13189.245} C_VEL
LIN {X 0,Y 361.861,Z 410.412,A -85,B 0,C 180,E1 -13191.574,E2 -13191.574} C_VEL
LIN {X 0,Y 361.827,Z 410.416,A -85,B 0,C 180,E1 -13192.977,E2 -13192.977} C_VEL
LIN {X 0,Y 361.807,Z 411.476,A -85,B 0,C 180,E1 -13194.671,E2 -13194.671} C_VEL
LIN {X 0,Y 361.722,Z 414.056,A -85,B 0,C 180,E1 -13197.042,E2 -13197.042} C_VEL
LIN {X 0,Y 361.556,Z 416.953,A -85,B 0,C 180,E1 -13199.643,E2 -13199.643} C_VEL
LIN {X 0,Y 361.3,Z 421.382,A -85,B 0,C 180,E1 -13203.482,E2 -13203.482} C_VEL
LIN {X 0,Y 361.014,Z 425.722,A -85,B 0,C 180,E1 -13207.086,E2 -13207.086} C_VEL
LIN {X 0,Y 360.924,Z 429.421,A -85,B 0,C 180,E1 -13209.993,E2 -13209.993} C_VEL
LIN {X 0,Y 364.349,Z 442.765,A -85,B 0,C 180,E1 -13210.698,E2 -13210.698} C_VEL
LIN {X 0,Y 366.843,Z 454.81,A -85,B 0,C 180,E1 -13211.513,E2 -13211.513} C_VEL
LIN {X 0,Y 367.585,Z 460.268,A -85,B 0,C 180,E1 -13211.935,E2 -13211.935} C_VEL
LIN {X 0,Y 366.613,Z 471.77,A -85,B 0,C 180,E1 -13212.858,E2 -13212.858} C_VEL
LIN {X 0,Y 365.719,Z 482.04,A -85,B 0,C 180,E1 -13213.915,E2 -13213.915} C_VEL
LIN {X 0,Y 364.741,Z 492.155,A -85,B 0,C 180,E1 -13215.208,E2 -13215.208} C_VEL
LIN {X 0,Y 363.646,Z 500.998,A -85,B 0,C 180,E1 -13216.59,E2 -13216.59} C_VEL
LIN {X 0,Y 362.697,Z 509.618,A -85,B 0,C 180,E1 -13218.261,E2 -13218.261} C_VEL
LIN {X 0,Y 361.895,Z 516.49,A -85,B 0,C 180,E1 -13219.934,E2 -13219.934} C_VEL
LIN {X 0,Y 361.227,Z 521.992,A -85,B 0,C 180,E1 -13221.61,E2 -13221.61} C_VEL
LIN {X 0,Y 360.845,Z 527.218,A -85,B 0,C 180,E1 -13223.705,E2 -13223.705} C_VEL
LIN {X 0,Y 360.558,Z 530.447,A -85,B 0,C 180,E1 -13225.528,E2 -13225.528} C_VEL
LIN {X 0,Y 360.418,Z 531.846,A -85,B 0,C 180,E1 -13226.646,E2 -13226.646} C_VEL
LIN {X 0,Y 360.353,Z 533.451,A -85,B 0,C 180,E1 -13228.883,E2 -13228.883} C_VEL
LIN {X 0,Y 360.361,Z 533.683,A -85,B 0,C 180,E1 -13230,E2 -13230} C_VEL
LIN {X 0,Y 360.353,Z 533.494,A -85,B 0,C 180,E1 -13231.118,E2 -13231.118} C_VEL
LIN {X 0,Y 360.413,Z 531.943,A -85,B 0,C 180,E1 -13233.354,E2 -13233.354} C_VEL
LIN {X 0,Y 360.551,Z 530.586,A -85,B 0,C 180,E1 -13234.472,E2 -13234.472} C_VEL
LIN {X 0,Y 360.79,Z 527.594,A -85,B 0,C 180,E1 -13236.217,E2 -13236.217} C_VEL
LIN {X 0,Y 361.112,Z 523.835,A -85,B 0,C 180,E1 -13237.83,E2 -13237.83} C_VEL
LIN {X 0,Y 361.619,Z 518.821,A -85,B 0,C 180,E1 -13239.509,E2 -13239.509} C_VEL
LIN {X 0,Y 362.3,Z 512.507,A -85,B 0,C 180,E1 -13241.185,E2 -13241.185} C_VEL
LIN {X 0,Y 363.241,Z 504.601,A -85,B 0,C 180,E1 -13242.856,E2 -13242.856} C_VEL
LIN {X 0,Y 364.432,Z 494.764,A -85,B 0,C 180,E1 -13244.519,E2 -13244.519} C_VEL
LIN {X 0,Y 365.381,Z 485.462,A -85,B 0,C 180,E1 -13245.783,E2 -13245.783} C_VEL
LIN {X 0,Y 366.378,Z 474.214,A -85,B 0,C 180,E1 -13247.01,E2 -13247.01} C_VEL
LIN {X 0,Y 367.424,Z 462.474,A -85,B 0,C 180,E1 -13248.01,E2 -13248.01} C_VEL
LIN {X 0,Y 367.521,Z 458.665,A -85,B 0,C 180,E1 -13248.288,E2 -13248.288} C_VEL
LIN {X 0,Y 365.135,Z 446.374,A -85,B 0,C 180,E1 -13249.185,E2 -13249.185} C_VEL
LIN {X 0,Y 362.086,Z 433.916,A -85,B 0,C 180,E1 -13249.899,E2 -13249.899} C_VEL
LIN {X 0,Y 360.933,Z 429.332,A -85,B 0,C 180,E1 -13250.143,E2 -13250.143} C_VEL
LIN {X 0,Y 361.134,Z 424.383,A -85,B 0,C 180,E1 -13254.122,E2 -13254.122} C_VEL
LIN {X 0,Y 361.375,Z 419.98,A -85,B 0,C 180,E1 -13257.824,E2 -13257.824} C_VEL
LIN {X 0,Y 361.617,Z 415.624,A -85,B 0,C 180,E1 -13261.651,E2 -13261.651} C_VEL
LIN {X 0,Y 361.722,Z 414.153,A -85,B 0,C 180,E1 -13262.963,E2 -13262.963} C_VEL
LIN {X 0,Y 361.084,Z 413.258,A -85,B 0,C 180,E1 -13263.882,E2 -13263.882} C_VEL
LIN {X 0,Y 358.263,Z 412.05,A -85,B 0,C 180,E1 -13265.384,E2 -13265.384} C_VEL
LIN {X 0,Y 355.873,Z 411.489,A -85,B 0,C 180,E1 -13266.606,E2 -13266.606} C_VEL
LIN {X 0,Y 354.865,Z 411.304,A -85,B 0,C 180,E1 -13267.552,E2 -13267.552} C_VEL
LIN {X 0,Y 354.793,Z 411.291,A -85,B 0,C 180,E1 -13267.872,E2 -13267.872} C_VEL
LIN {X 0,Y 354.79,Z 411.29,A -85,B 0,C 180,E1 -13271.172,E2 -13271.172} C_VEL
LIN {X 0,Y 354.811,Z 411.289,A -85,B 0,C 180,E1 -13274.514,E2 -13274.514} C_VEL
LIN {X 0,Y 354.797,Z 411.287,A -85,B 0,C 180,E1 -13277.663,E2 -13277.663} C_VEL
LIN {X 0,Y 354.817,Z 411.29,A -85,B 0,C 180,E1 -13280.666,E2 -13280.666} C_VEL
LIN {X 0,Y 354.825,Z 411.287,A -85,B 0,C 180,E1 -13284.301,E2 -13284.301} C_VEL
LIN {X 0,Y 354.789,Z 411.288,A -85,B 0,C 180,E1 -13287.667,E2 -13287.667} C_VEL
LIN {X 0,Y 354.831,Z 411.286,A -85,B 0,C 180,E1 -13290.633,E2 -13290.633} C_VEL
LIN {X 0,Y 354.902,Z 411.278,A -85,B 0,C 180,E1 -13294.173,E2 -13294.173} C_VEL
LIN {X 0,Y 354.837,Z 411.284,A -85,B 0,C 180,E1 -13297.894,E2 -13297.894} C_VEL
LIN {X 0,Y 354.925,Z 411.274,A -85,B 0,C 180,E1 -13301.892,E2 -13301.892} C_VEL
LIN {X 0,Y 354.945,Z 411.273,A -85,B 0,C 180,E1 -13305.981,E2 -13305.981} C_VEL
LIN {X 0,Y 354.981,Z 411.267,A -85,B 0,C 180,E1 -13309.736,E2 -13309.736} C_VEL
LIN {X 0,Y 355.117,Z 411.252,A -85,B 0,C 180,E1 -13312.037,E2 -13312.037} C_VEL
LIN {X 0,Y 355.095,Z 411.252,A -85,B 0,C 180,E1 -13314.321,E2 -13314.321} C_VEL
LIN {X 0,Y 355.246,Z 411.235,A -85,B 0,C 180,E1 -13317.732,E2 -13317.732} C_VEL
LIN {X 0,Y 355.399,Z 411.216,A -85,B 0,C 180,E1 -13320,E2 -13320} C_VEL
LIN {X 0,Y 355.247,Z 411.232,A -85,B 0,C 180,E1 -13322.268,E2 -13322.268} C_VEL
LIN {X 0,Y 355.141,Z 411.244,A -85,B 0,C 180,E1 -13326.819,E2 -13326.819} C_VEL
LIN {X 0,Y 355.02,Z 411.26,A -85,B 0,C 180,E1 -13329.112,E2 -13329.112} C_VEL
LIN {X 0,Y 354.929,Z 411.27,A -85,B 0,C 180,E1 -13332.581,E2 -13332.581} C_VEL
LIN {X 0,Y 354.893,Z 411.276,A -85,B 0,C 180,E1 -13336.096,E2 -13336.096} C_VEL
LIN {X 0,Y 354.904,Z 411.273,A -85,B 0,C 180,E1 -13338.472,E2 -13338.472} C_VEL
LIN {X 0,Y 354.837,Z 411.282,A -85,B 0,C 180,E1 -13342.106,E2 -13342.106} C_VEL
LIN {X 0,Y 354.901,Z 411.275,A -85,B 0,C 180,E1 -13345.827,E2 -13345.827} C_VEL
LIN {X 0,Y 354.82,Z 411.286,A -85,B 0,C 180,E1 -13349.682,E2 -13349.682} C_VEL
LIN {X 0,Y 354.808,Z 411.286,A -85,B 0,C 180,E1 -13353.702,E2 -13353.702} C_VEL
LIN {X 0,Y 354.801,Z 411.287,A -85,B 0,C 180,E1 -13356.459,E2 -13356.459} C_VEL
LIN {X 0,Y 354.826,Z 411.286,A -85,B 0,C 180,E1 -13359.424,E2 -13359.424} C_VEL
